KUKA KRL program: MyProgram_268().src

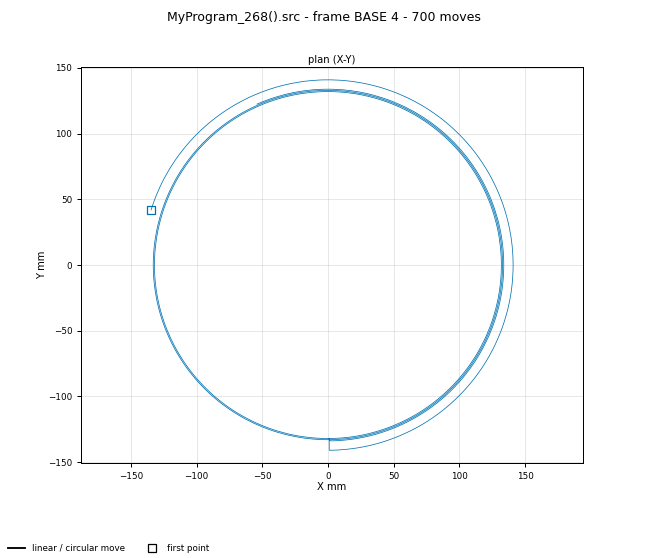
[picture p0: tool path of MyProgram_268().src in frame BASE 4, 700 of 700 moves have a stored position in this frame; points joined in program order, loops and branches not executed]
&ACCESS RVP
&REL 1
&PARAM TEMPLATE = C:\KRC\Roboter\Template\vorgabe
&PARAM EDITMASK = *
DEF MyProgram_268()
; ---- Setting reference (Base) ----
$BASE = BASE_DATA[4]

; --------------------------
; ---- Setting tool (TCP) ----
$TOOL = TOOL_DATA[3]
; --------------------------

$VEL.CP = VEL_APROX_PRINT
Startdeposition()
$VEL.CP = VEL_PRINT
LIN {X -134.5942,Y 41.9312,Z 169,A 163.5765,B 9.595,C 0.2023,E1 9.4446,E2 287.9092} C_DIS
LIN {X -133.5256,Y 45.2188,Z 169,A 161.9808,B 9.595,C 0.2018,E1 9.446,E2 289.5276} C_DIS
LIN {X -132.144,Y 49.1059,Z 169,A 160.3051,B 9.5951,C 0.1972,E1 9.4476,E2 291.2013} C_DIS
LIN {X -130.5039,Y 53.3146,Z 169,A 158.5648,B 9.5953,C 0.1905,E1 9.4494,E2 292.9277} C_DIS
LIN {X -129.1483,Y 56.5189,Z 169,A 157.1411,B 9.5953,C 0.1868,E1 9.451,E2 294.3512} C_DIS
LIN {X -127.8004,Y 59.5017,Z 169,A 155.7818,B 9.5953,C 0.1838,E1 9.4525,E2 295.7126} C_DIS
LIN {X -126.3044,Y 62.6142,Z 169,A 154.3586,B 9.5955,C 0.1804,E1 9.4543,E2 297.1368} C_DIS
LIN {X -124.5762,Y 65.9871,Z 169,A 152.7987,B 9.5955,C 0.1768,E1 9.4563,E2 298.6975} C_DIS
LIN {X -122.6643,Y 69.4801,Z 169,A 151.0806,B 9.5955,C 0.1745,E1 9.4586,E2 300.4266} C_DIS
LIN {X -120.481,Y 73.2001,Z 169,A 149.3244,B 9.5956,C 0.1701,E1 9.4612,E2 302.1813} C_DIS
LIN {X -118.1952,Y 76.8358,Z 169,A 147.5146,B 9.5957,C 0.167,E1 9.4639,E2 303.9974} C_DIS
LIN {X -115.5599,Y 80.7454,Z 169,A 145.5711,B 9.5957,C 0.1628,E1 9.467,E2 305.9422} C_DIS
LIN {X -113.0324,Y 84.2467,Z 169,A 143.81,B 9.5958,C 0.1587,E1 9.4699,E2 307.7022} C_DIS
LIN {X -110.5027,Y 87.5391,Z 169,A 142.0533,B 9.5958,C 0.1561,E1 9.4729,E2 309.466} C_DIS
LIN {X -107.5268,Y 91.1694,Z 169,A 140.2431,B 9.596,C 0.15,E1 9.4761,E2 311.2619} C_DIS
LIN {X -104.992,Y 94.0771,Z 169,A 138.5981,B 9.596,C 0.1479,E1 9.4792,E2 312.915} C_DIS
LIN {X -102.0667,Y 97.2434,Z 169,A 136.8251,B 9.596,C 0.1446,E1 9.4825,E2 314.6888} C_DIS
LIN {X -99.0916,Y 100.2738,Z 169,A 135.045,B 9.5961,C 0.142,E1 9.4861,E2 316.474} C_DIS
LIN {X -95.7403,Y 103.4786,Z 169,A 133.1345,B 9.5961,C 0.1386,E1 9.4899,E2 318.3859} C_DIS
LIN {X -92.5309,Y 106.3574,Z 169,A 131.3797,B 9.5961,C 0.1352,E1 9.4936,E2 320.1393} C_DIS
LIN {X -89.2875,Y 109.0944,Z 169,A 129.6507,B 9.5962,C 0.1321,E1 9.4973,E2 321.8672} C_DIS
LIN {X -85.7732,Y 111.8785,Z 169,A 127.7709,B 9.5962,C 0.1298,E1 9.5015,E2 323.7525} C_DIS
LIN {X -81.9982,Y 114.674,Z 169,A 125.8885,B 9.5963,C 0.126,E1 9.5057,E2 325.6297} C_DIS
LIN {X -78.322,Y 117.2156,Z 169,A 124.0447,B 9.5963,C 0.1235,E1 9.51,E2 327.4753} C_DIS
LIN {X -74.6865,Y 119.5651,Z 169,A 122.2899,B 9.5963,C 0.1206,E1 9.5141,E2 329.2279} C_DIS
LIN {X -70.9951,Y 121.7937,Z 169,A 120.4792,B 9.5964,C 0.1191,E1 9.5185,E2 331.0444} C_DIS
LIN {X -67.2172,Y 123.9185,Z 169,A 118.6942,B 9.5964,C 0.117,E1 9.5228,E2 332.8309} C_DIS
LIN {X -63.389,Y 125.9186,Z 169,A 117.039,B 9.5964,C 0.1126,E1 9.5269,E2 334.4719} C_DIS
LIN {X -60.2838,Y 127.434,Z 169,A 115.6266,B 9.5965,C 0.111,E1 9.5305,E2 335.8842} C_DIS
LIN {X -57.1208,Y 128.8826,Z 169,A 114.2055,B 9.5965,C 0.1094,E1 9.5341,E2 337.305} C_DIS
LIN {X -53.3354,Y 130.4955,Z 169,A 112.4278,B 9.5965,C 0.1095,E1 9.5387,E2 339.0947} C_DIS
LIN {X -49.779,Y 131.8919,Z 169,A 110.9649,B 9.5965,C 0.1061,E1 9.5425,E2 340.5449} C_DIS
LIN {X -46.5347,Y 133.0713,Z 169,A 109.5024,B 9.5965,C 0.1058,E1 9.5463,E2 342.0139} C_DIS
LIN {X -42.5768,Y 134.3899,Z 169,A 107.8494,B 9.5965,C 0.1034,E1 9.5507,E2 343.6603} C_DIS
LIN {X -39.2696,Y 135.3933,Z 169,A 106.4388,B 9.5966,C 0.1023,E1 9.5545,E2 345.0706} C_DIS
LIN {X -35.282,Y 136.4877,Z 169,A 104.6517,B 9.5966,C 0.1032,E1 9.5593,E2 346.87} C_DIS
LIN {X -31.7318,Y 137.3556,Z 169,A 103.2097,B 9.5966,C 0.1012,E1 9.5632,E2 348.3056} C_DIS
LIN {X -27.4911,Y 138.2678,Z 169,A 101.5074,B 9.5966,C 0.0989,E1 9.5679,E2 349.9991} C_DIS
LIN {X -24.1085,Y 138.8981,Z 169,A 100.0991,B 9.5966,C 0.0984,E1 9.5717,E2 351.4079} C_DIS
LIN {X -20.708,Y 139.4459,Z 169,A 98.674,B 9.5966,C 0.0982,E1 9.5757,E2 352.8352} C_DIS
LIN {X -17.26,Y 139.9135,Z 169,A 97.1242,B 9.5966,C 0.1004,E1 9.58,E2 354.4012} C_DIS
LIN {X -12.7769,Y 140.3946,Z 169,A 95.4449,B 9.5966,C 0.0967,E1 9.5846,E2 356.0603} C_DIS
LIN {X -9.3326,Y 140.6654,Z 169,A 94.0962,B 9.5966,C 0.0952,E1 9.5884,E2 357.4014} C_DIS
LIN {X -6.258,Y 140.8362,Z 169,A 92.7456,B 9.5966,C 0.097,E1 9.5922,E2 358.7638} C_DIS
LIN {X -2.4077,Y 140.9526,Z 169,A 91.1279,B 9.5966,C 0.0979,E1 9.5967,E2 360.3872} C_DIS
LIN {X 2.3955,Y 140.9528,Z 169,A 89.2128,B 9.5966,C 0.0972,E1 9.602,E2 362.2968} C_DIS
LIN {X 6.234,Y 140.8372,Z 169,A 87.6868,B 9.5966,C 0.0965,E1 9.6063,E2 363.8178} C_DIS
LIN {X 9.3191,Y 140.6662,Z 169,A 86.4564,B 9.5966,C 0.0962,E1 9.6097,E2 365.0445} C_DIS
LIN {X 12.7648,Y 140.3957,Z 169,A 84.9273,B 9.5966,C 0.0991,E1 9.614,E2 366.5887} C_DIS
LIN {X 17.2433,Y 139.9155,Z 169,A 83.2176,B 9.5966,C 0.0971,E1 9.6187,E2 368.2825} C_DIS
LIN {X 20.6777,Y 139.4502,Z 169,A 81.8119,B 9.5966,C 0.0976,E1 9.6226,E2 369.6875} C_DIS
LIN {X 23.453,Y 139.0086,Z 169,A 80.6674,B 9.5966,C 0.0981,E1 9.6257,E2 370.8318} C_DIS
LIN {X 26.8316,Y 138.3964,Z 169,A 79.1656,B 9.5966,C 0.1011,E1 9.6299,E2 372.3466} C_DIS
LIN {X 31.5211,Y 137.4037,Z 169,A 77.3288,B 9.5966,C 0.0999,E1 9.6349,E2 374.169} C_DIS
LIN {X 35.2505,Y 136.4957,Z 169,A 75.782,B 9.5966,C 0.1006,E1 9.6391,E2 375.7137} C_DIS
LIN {X 38.615,Y 135.5827,Z 169,A 74.3639,B 9.5966,C 0.1017,E1 9.6429,E2 377.1318} C_DIS
LIN {X 41.9329,Y 134.5936,Z 169,A 72.9765,B 9.5966,C 0.1024,E1 9.6466,E2 378.5164} C_DIS
LIN {X 45.2213,Y 133.5247,Z 169,A 71.4108,B 9.5966,C 0.1072,E1 9.6508,E2 380.1023} C_DIS
LIN {X 49.1122,Y 132.1417,Z 169,A 69.7678,B 9.5966,C 0.1081,E1 9.6551,E2 381.7406} C_DIS
LIN {X 53.3187,Y 130.5023,Z 169,A 68.0634,B 9.5966,C 0.1071,E1 9.6594,E2 383.4284} C_DIS
LIN {X 56.5128,Y 129.1509,Z 169,A 66.6736,B 9.5966,C 0.1082,E1 9.663,E2 384.8156} C_DIS
LIN {X 59.4777,Y 127.8115,Z 169,A 65.3498,B 9.5966,C 0.1098,E1 9.6664,E2 386.1396} C_DIS
LIN {X 62.5803,Y 126.3212,Z 169,A 63.9205,B 9.5965,C 0.1122,E1 9.67,E2 387.5727} C_DIS
LIN {X 66.4245,Y 124.3453,Z 169,A 62.2133,B 9.5965,C 0.1134,E1 9.6742,E2 389.2738} C_DIS
LIN {X 69.7802,Y 122.4931,Z 169,A 60.5878,B 9.5965,C 0.1171,E1 9.6782,E2 390.9079} C_DIS
LIN {X 73.5011,Y 120.2975,Z 169,A 58.8315,B 9.5965,C 0.1197,E1 9.6824,E2 392.6644} C_DIS
LIN {X 77.5895,Y 117.7018,Z 169,A 56.8943,B 9.5964,C 0.1221,E1 9.6869,E2 394.598} C_DIS
LIN {X 81.1458,Y 115.2788,Z 169,A 55.1544,B 9.5964,C 0.1247,E1 9.6909,E2 396.3371} C_DIS
LIN {X 84.6708,Y 112.7155,Z 169,A 53.4186,B 9.5964,C 0.1269,E1 9.6948,E2 398.0687} C_DIS
LIN {X 88.0894,Y 110.0647,Z 169,A 51.6799,B 9.5963,C 0.1296,E1 9.6986,E2 399.8054} C_DIS
LIN {X 91.4161,Y 107.317,Z 169,A 49.9188,B 9.5963,C 0.1329,E1 9.7024,E2 401.5679} C_DIS
LIN {X 94.6711,Y 104.4568,Z 169,A 48.1785,B 9.5962,C 0.1358,E1 9.706,E2 403.306} C_DIS
LIN {X 97.836,Y 101.4989,Z 169,A 46.4418,B 9.5962,C 0.1387,E1 9.7095,E2 405.0403} C_DIS
LIN {X 100.8967,Y 98.4571,Z 169,A 44.7252,B 9.5962,C 0.1414,E1 9.7129,E2 406.7527} C_DIS
LIN {X 103.8624,Y 95.3229,Z 169,A 43.0024,B 9.5961,C 0.1444,E1 9.7161,E2 408.4723} C_DIS
LIN {X 106.7472,Y 92.0808,Z 169,A 41.2219,B 9.5961,C 0.1486,E1 9.7194,E2 410.2556} C_DIS
LIN {X 109.5218,Y 88.7632,Z 169,A 39.4703,B 9.5959,C 0.1524,E1 9.7225,E2 412.0072} C_DIS
LIN {X 112.187,Y 85.3699,Z 169,A 37.7746,B 9.5959,C 0.155,E1 9.7254,E2 413.6964} C_DIS
LIN {X 114.7571,Y 81.882,Z 169,A 36.0512,B 9.5959,C 0.1582,E1 9.7282,E2 415.4159} C_DIS
LIN {X 117.2128,Y 78.3262,Z 169,A 34.2819,B 9.5958,C 0.1627,E1 9.731,E2 417.1878} C_DIS
LIN {X 119.555,Y 74.7028,Z 169,A 32.5697,B 9.5958,C 0.1659,E1 9.7336,E2 418.8957} C_DIS
LIN {X 121.7798,Y 71.0191,Z 169,A 30.7924,B 9.5956,C 0.171,E1 9.7361,E2 420.6776} C_DIS
LIN {X 123.9192,Y 67.2159,Z 169,A 29.0406,B 9.5956,C 0.1749,E1 9.7385,E2 422.4277} C_DIS
LIN {X 125.7674,Y 63.686,Z 169,A 27.522,B 9.5956,C 0.1766,E1 9.7404,E2 423.9344} C_DIS
LIN {X 127.4446,Y 60.2617,Z 169,A 26.0271,B 9.5955,C 0.1793,E1 9.7422,E2 425.4234} C_DIS
LIN {X 128.8415,Y 57.2127,Z 169,A 24.6768,B 9.5955,C 0.1826,E1 9.7438,E2 426.7729} C_DIS
LIN {X 130.4933,Y 53.341,Z 169,A 22.9043,B 9.5953,C 0.1887,E1 9.7457,E2 428.5546} C_DIS
LIN {X 131.8908,Y 49.782,Z 169,A 21.4593,B 9.5953,C 0.1902,E1 9.7471,E2 429.9867} C_DIS
LIN {X 133.3051,Y 45.8604,Z 169,A 19.7974,B 9.5952,C 0.194,E1 9.7487,E2 431.6457} C_DIS
LIN {X 134.3891,Y 42.5794,Z 169,A 18.4143,B 9.5952,C 0.1974,E1 9.7499,E2 433.0272} C_DIS
LIN {X 135.3924,Y 39.2725,Z 169,A 17.0291,B 9.5951,C 0.2008,E1 9.751,E2 434.411} C_DIS
LIN {X 136.4894,Y 35.2754,Z 169,A 15.2736,B 9.5949,C 0.2073,E1 9.7522,E2 436.177} C_DIS
LIN {X 137.4032,Y 31.5233,Z 169,A 13.8229,B 9.5949,C 0.2088,E1 9.7532,E2 437.6137} C_DIS
LIN {X 138.267,Y 27.495,Z 169,A 12.1816,B 9.5949,C 0.2127,E1 9.7541,E2 439.2522} C_DIS
LIN {X 138.8977,Y 24.1109,Z 169,A 10.8273,B 9.5947,C 0.2156,E1 9.7548,E2 440.6019} C_DIS
LIN {X 139.3437,Y 21.3717,Z 169,A 9.6887,B 9.5947,C 0.2191,E1 9.7553,E2 441.7429} C_DIS
LIN {X 139.8288,Y 17.9286,Z 169,A 8.1786,B 9.5945,C 0.2256,E1 9.7558,E2 443.2667} C_DIS
LIN {X 140.295,Y 13.8137,Z 169,A 6.6283,B 9.5945,C 0.2272,E1 9.7563,E2 444.8015} C_DIS
LIN {X 140.5909,Y 10.374,Z 169,A 5.2517,B 9.5944,C 0.2306,E1 9.7566,E2 446.1759} C_DIS
LIN {X 140.8029,Y 6.9279,Z 169,A 3.8772,B 9.5944,C 0.234,E1 9.7568,E2 447.548} C_DIS
LIN {X 140.931,Y 3.4756,Z 169,A 2.5047,B 9.5942,C 0.2373,E1 9.7569,E2 448.9178} C_DIS
LIN {X 140.9775,Y -0.0022,Z 169,A 0.8866,B 9.594,C 0.2465,E1 9.7569,E2 450.5638} C_DIS
LIN {X 140.9022,Y -4.5117,Z 169,A -0.6897,B 9.594,C 0.2455,E1 9.7569,E2 452.1086} C_DIS
LIN {X 140.7496,Y -7.9654,Z 169,A -2.0369,B 9.594,C 0.2481,E1 9.7567,E2 453.4496} C_DIS
LIN {X 140.5425,Y -11.0367,Z 169,A -3.3352,B 9.5938,C 0.2529,E1 9.7564,E2 454.7554} C_DIS
LIN {X 140.1868,Y -14.8698,Z 169,A -4.87,B 9.5938,C 0.2567,E1 9.756,E2 456.2878} C_DIS
LIN {X 139.693,Y -18.9651,Z 169,A -6.5053,B 9.5936,C 0.2606,E1 9.7554,E2 457.9195} C_DIS
LIN {X 139.1873,Y -22.3816,Z 169,A -7.9131,B 9.5936,C 0.2648,E1 9.7548,E2 459.3294} C_DIS
LIN {X 138.5947,Y -25.7943,Z 169,A -9.2934,B 9.5934,C 0.2681,E1 9.7541,E2 460.7075} C_DIS
LIN {X 137.8647,Y -29.4408,Z 169,A -10.8555,B 9.5933,C 0.2737,E1 9.7532,E2 462.2777} C_DIS
LIN {X 137.0081,Y -33.1984,Z 169,A -12.3595,B 9.5932,C 0.2767,E1 9.7523,E2 463.7752} C_DIS
LIN {X 136.0578,Y -36.9049,Z 169,A -13.8478,B 9.5932,C 0.2794,E1 9.7512,E2 465.2565} C_DIS
LIN {X 135.1126,Y -40.2284,Z 169,A -15.2331,B 9.593,C 0.2829,E1 9.7501,E2 466.6408} C_DIS
LIN {X 134.1854,Y -43.2169,Z 169,A -16.5209,B 9.5929,C 0.2869,E1 9.749,E2 467.9321} C_DIS
LIN {X 132.7343,Y -47.487,Z 169,A -18.2601,B 9.5929,C 0.2897,E1 9.7475,E2 469.661} C_DIS
LIN {X 131.2801,Y -51.3705,Z 169,A -19.9923,B 9.5926,C 0.2955,E1 9.7457,E2 471.4011} C_DIS
LIN {X 129.8366,Y -54.9196,Z 169,A -21.4938,B 9.5926,C 0.2984,E1 9.7441,E2 472.8971} C_DIS
LIN {X 128.532,Y -57.9047,Z 169,A -22.7978,B 9.5925,C 0.3015,E1 9.7427,E2 474.1998} C_DIS
LIN {X 127.0634,Y -61.0594,Z 169,A -24.1927,B 9.5923,C 0.3048,E1 9.741,E2 475.5938} C_DIS
LIN {X 125.3754,Y -64.4561,Z 169,A -25.7756,B 9.5922,C 0.3099,E1 9.739,E2 477.1837} C_DIS
LIN {X 123.2498,Y -68.435,Z 169,A -27.5651,B 9.5921,C 0.3136,E1 9.7366,E2 478.9695} C_DIS
LIN {X 121.0914,Y -72.1853,Z 169,A -29.3064,B 9.5919,C 0.3177,E1 9.7342,E2 480.7104} C_DIS
LIN {X 118.9256,Y -75.7012,Z 169,A -31.0146,B 9.5918,C 0.3227,E1 9.7316,E2 482.4243} C_DIS
LIN {X 116.4553,Y -79.4491,Z 169,A -32.8335,B 9.5916,C 0.327,E1 9.7288,E2 484.2444} C_DIS
LIN {X 113.7961,Y -83.2128,Z 169,A -34.6594,B 9.5916,C 0.3305,E1 9.7258,E2 486.0662} C_DIS
LIN {X 111.1913,Y -86.663,Z 169,A -36.4151,B 9.5914,C 0.3346,E1 9.7228,E2 487.8235} C_DIS
LIN {X 108.4264,Y -90.0977,Z 169,A -38.158,B 9.5913,C 0.3376,E1 9.7198,E2 489.5619} C_DIS
LIN {X 105.6201,Y -93.3715,Z 169,A -39.8759,B 9.5911,C 0.3407,E1 9.7166,E2 491.277} C_DIS
LIN {X 102.7099,Y -96.5637,Z 169,A -41.6013,B 9.5911,C 0.3439,E1 9.7133,E2 493.0003} C_DIS
LIN {X 99.6849,Y -99.6843,Z 169,A -43.3281,B 9.5909,C 0.3467,E1 9.71,E2 494.7238} C_DIS
LIN {X 96.5855,Y -102.6894,Z 169,A -45.0601,B 9.5909,C 0.3499,E1 9.7065,E2 496.4546} C_DIS
LIN {X 93.3954,Y -105.5989,Z 169,A -46.8058,B 9.5907,C 0.3532,E1 9.7029,E2 498.2008} C_DIS
LIN {X 90.0987,Y -108.4256,Z 169,A -48.5608,B 9.5906,C 0.3565,E1 9.6991,E2 499.9563} C_DIS
LIN {X 86.7378,Y -111.1331,Z 169,A -50.3042,B 9.5905,C 0.3595,E1 9.6953,E2 501.7} C_DIS
LIN {X 83.2951,Y -113.7356,Z 169,A -52.0622,B 9.5903,C 0.3629,E1 9.6914,E2 503.4602} C_DIS
LIN {X 79.773,Y -116.2329,Z 169,A -53.7663,B 9.5903,C 0.3647,E1 9.6875,E2 505.1593} C_DIS
LIN {X 76.1662,Y -118.6279,Z 169,A -55.5425,B 9.5901,C 0.3681,E1 9.6833,E2 506.9393} C_DIS
LIN {X 72.5117,Y -120.8968,Z 169,A -57.2905,B 9.5901,C 0.3709,E1 9.6791,E2 508.6889} C_DIS
LIN {X 68.7803,Y -123.0578,Z 169,A -58.998,B 9.59,C 0.3726,E1 9.675,E2 510.392} C_DIS
LIN {X 65.3914,Y -124.889,Z 169,A -60.5053,B 9.59,C 0.3735,E1 9.6713,E2 511.893} C_DIS
LIN {X 61.8369,Y -126.6879,Z 169,A -62.0901,B 9.5899,C 0.375,E1 9.6673,E2 513.4747} C_DIS
LIN {X 58.733,Y -128.1559,Z 169,A -63.4717,B 9.5899,C 0.3766,E1 9.6639,E2 514.8557} C_DIS
LIN {X 55.6106,Y -129.541,Z 169,A -64.8591,B 9.5898,C 0.3783,E1 9.6603,E2 516.2441} C_DIS
LIN {X 51.8495,Y -131.0939,Z 169,A -66.6301,B 9.5896,C 0.383,E1 9.6557,E2 518.0318} C_DIS
LIN {X 47.5078,Y -132.7268,Z 169,A -68.3666,B 9.5896,C 0.3817,E1 9.6512,E2 519.7503} C_DIS
LIN {X 44.2426,Y -133.8506,Z 169,A -69.762,B 9.5896,C 0.383,E1 9.6475,E2 521.1456} C_DIS
LIN {X 40.9236,Y -134.9026,Z 169,A -71.1692,B 9.5896,C 0.3842,E1 9.6437,E2 522.5528} C_DIS
LIN {X 37.6033,Y -135.8656,Z 169,A -72.6736,B 9.5894,C 0.3877,E1 9.6396,E2 524.0714} C_DIS
LIN {X 33.2171,Y -137.0036,Z 169,A -74.4025,B 9.5894,C 0.3867,E1 9.635,E2 525.7867} C_DIS
LIN {X 29.857,Y -137.7749,Z 169,A -75.8844,B 9.5894,C 0.3896,E1 9.6309,E2 527.2801} C_DIS
LIN {X 25.821,Y -138.5896,Z 169,A -77.4557,B 9.5894,C 0.3884,E1 9.6266,E2 528.8392} C_DIS
LIN {X 22.4208,Y -139.1808,Z 169,A -78.8725,B 9.5894,C 0.3896,E1 9.6227,E2 530.2587} C_DIS
LIN {X 18.9812,Y -139.6909,Z 169,A -80.2838,B 9.5893,C 0.3903,E1 9.6188,E2 531.6707} C_DIS
LIN {X 14.868,Y -140.187,Z 169,A -81.982,B 9.5893,C 0.3914,E1 9.6141,E2 533.3717} C_DIS
LIN {X 11.1093,Y -140.5367,Z 169,A -83.5081,B 9.5893,C 0.3918,E1 9.6099,E2 534.8976} C_DIS
LIN {X 7.9782,Y -140.7489,Z 169,A -84.7464,B 9.5893,C 0.3914,E1 9.6064,E2 536.1317} C_DIS
LIN {X 4.5253,Y -140.9018,Z 169,A -86.2616,B 9.5891,C 0.3941,E1 9.6022,E2 537.6621} C_DIS
LIN {X 1.0246,Y -140.9657,Z 169,A -87.164,B 9.5896,C 0.3829,E1 9.5998,E2 538.4966} C_DIS
Enddeposition()
LIN {X 0.9572,Y -132.0209,Z 170,A -87.7415,B 9.9605,C 0.3252,E1 9.9679,E2 538.6917} C_DIS
Startdeposition()
$VEL.CP = VEL_PRINT
LIN {X 3.7904,Y -131.9708,Z 170,A -86.115,B 9.9607,C 0.3165,E1 9.9726,E2 537.0162} C_DIS
LIN {X 8.0863,Y -131.7772,Z 170,A -84.3027,B 9.9607,C 0.3172,E1 9.9776,E2 535.2096} C_DIS
LIN {X 11.8723,Y -131.4923,Z 170,A -82.5093,B 9.9608,C 0.3134,E1 9.9827,E2 533.3975} C_DIS
LIN {X 16.16,Y -131.0333,Z 170,A -80.6725,B 9.9608,C 0.3134,E1 9.9878,E2 531.5638} C_DIS
LIN {X 19.3657,Y -130.5988,Z 170,A -79.4051,B 9.9608,C 0.3155,E1 9.9912,E2 530.3123} C_DIS
LIN {X 23.1047,Y -129.9876,Z 170,A -77.7513,B 9.9608,C 0.3143,E1 9.9958,E2 528.6562} C_DIS
LIN {X 26.3031,Y -129.3782,Z 170,A -76.2726,B 9.9608,C 0.3119,E1 9.9999,E2 527.1686} C_DIS
LIN {X 30.5034,Y -128.4535,Z 170,A -74.482,B 9.9608,C 0.3121,E1 10.0047,E2 525.386} C_DIS
LIN {X 33.6448,Y -127.6665,Z 170,A -73.0844,B 9.9609,C 0.3111,E1 10.0085,E2 523.9884} C_DIS
LIN {X 36.7643,Y -126.8032,Z 170,A -71.5383,B 9.9611,C 0.3067,E1 10.0127,E2 522.4238} C_DIS
LIN {X 41.3922,Y -125.3688,Z 170,A -69.4899,B 9.9611,C 0.3058,E1 10.0181,E2 520.3805} C_DIS
LIN {X 44.9083,Y -124.1523,Z 170,A -67.937,B 9.9611,C 0.3054,E1 10.0222,E2 518.834} C_DIS
LIN {X 48.7091,Y -122.7128,Z 170,A -66.077,B 9.9612,C 0.3012,E1 10.0271,E2 516.9609} C_DIS
LIN {X 52.0153,Y -121.3469,Z 170,A -64.698,B 9.9612,C 0.3031,E1 10.0306,E2 515.6017} C_DIS
LIN {X 54.9745,Y -120.0355,Z 170,A -63.3038,B 9.9612,C 0.3015,E1 10.0341,E2 514.2077} C_DIS
LIN {X 57.9001,Y -118.6524,Z 170,A -61.8704,B 9.9612,C 0.2989,E1 10.0377,E2 512.7696} C_DIS
LIN {X 60.8063,Y -117.19,Z 170,A -60.4164,B 9.9614,C 0.2959,E1 10.0414,E2 511.3092} C_DIS
LIN {X 64.1291,Y -115.4059,Z 170,A -58.8145,B 9.9614,C 0.2943,E1 10.0453,E2 509.7102} C_DIS
LIN {X 67.8372,Y -113.2661,Z 170,A -57.0334,B 9.9614,C 0.2931,E1 10.0496,E2 507.9367} C_DIS
LIN {X 70.629,Y -111.5464,Z 170,A -55.5169,B 9.9616,C 0.2886,E1 10.0532,E2 506.4074} C_DIS
LIN {X 73.8128,Y -109.4657,Z 170,A -53.8877,B 9.9616,C 0.2862,E1 10.057,E2 504.7793} C_DIS
LIN {X 77.3447,Y -106.9993,Z 170,A -52.1417,B 9.9616,C 0.2857,E1 10.0609,E2 503.0466} C_DIS
LIN {X 80.1576,Y -104.9084,Z 170,A -50.5419,B 9.9618,C 0.2811,E1 10.0645,E2 501.4358} C_DIS
LIN {X 83.542,Y -102.2338,Z 170,A -48.6838,B 9.9618,C 0.2778,E1 10.0685,E2 499.5775} C_DIS
LIN {X 86.8446,Y -99.4436,Z 170,A -46.8696,B 9.962,C 0.2755,E1 10.0724,E2 497.7691} C_DIS
LIN {X 89.847,Y -96.7397,Z 170,A -45.1313,B 9.962,C 0.2723,E1 10.076,E2 496.0308} C_DIS
LIN {X 92.7363,Y -93.9743,Z 170,A -43.3386,B 9.9622,C 0.2673,E1 10.0796,E2 494.2294} C_DIS
LIN {X 95.6179,Y -91.0401,Z 170,A -41.661,B 9.9622,C 0.2659,E1 10.0828,E2 492.5631} C_DIS
LIN {X 98.3647,Y -88.0648,Z 170,A -39.8809,B 9.9623,C 0.2614,E1 10.0861,E2 490.7784} C_DIS
LIN {X 100.996,Y -85.0345,Z 170,A -38.1028,B 9.9625,C 0.2566,E1 10.0894,E2 488.9939} C_DIS
LIN {X 103.9098,Y -81.4481,Z 170,A -36.2159,B 9.9625,C 0.2547,E1 10.0926,E2 487.1194} C_DIS
LIN {X 106.375,Y -78.2009,Z 170,A -34.5164,B 9.9625,C 0.2521,E1 10.0955,E2 485.4266} C_DIS
LIN {X 108.2546,Y -75.5778,Z 170,A -33.0352,B 9.9627,C 0.2467,E1 10.0979,E2 483.934} C_DIS
LIN {X 110.6681,Y -71.9972,Z 170,A -31.1834,B 9.9628,C 0.2426,E1 10.1007,E2 482.0829} C_DIS
LIN {X 112.694,Y -68.7836,Z 170,A -29.5428,B 9.9628,C 0.2386,E1 10.1031,E2 480.4414} C_DIS
LIN {X 114.8835,Y -65.0613,Z 170,A -27.7988,B 9.9629,C 0.2368,E1 10.1056,E2 478.7113} C_DIS
LIN {X 116.4391,Y -62.2338,Z 170,A -26.2814,B 9.9631,C 0.2304,E1 10.1076,E2 477.1781} C_DIS
LIN {X 118.172,Y -58.8739,Z 170,A -24.8109,B 9.9631,C 0.2301,E1 10.1094,E2 475.7266} C_DIS
LIN {X 119.5747,Y -55.9711,Z 170,A -23.4316,B 9.9631,C 0.2268,E1 10.1111,E2 474.3482} C_DIS
LIN {X 120.9038,Y -53.0403,Z 170,A -22.0317,B 9.9633,C 0.2229,E1 10.1127,E2 472.9464} C_DIS
LIN {X 122.3784,Y -49.5386,Z 170,A -20.6011,B 9.9633,C 0.2236,E1 10.1142,E2 471.5404} C_DIS
LIN {X 123.3769,Y -47.0023,Z 170,A -19.1123,B 9.9635,C 0.2131,E1 10.1157,E2 470.0132} C_DIS
LIN {X 124.8489,Y -42.9345,Z 170,A -17.403,B 9.9635,C 0.2119,E1 10.1173,E2 468.3223} C_DIS
LIN {X 126.0377,Y -39.3132,Z 170,A -15.6421,B 9.9636,C 0.2046,E1 10.1188,E2 466.5467} C_DIS
LIN {X 126.9502,Y -36.2591,Z 170,A -14.2692,B 9.9637,C 0.201,E1 10.1199,E2 465.1736} C_DIS
LIN {X 127.7953,Y -33.1572,Z 170,A -13.0332,B 9.9637,C 0.2008,E1 10.1207,E2 463.9554} C_DIS
LIN {X 128.5625,Y -30.0449,Z 170,A -11.6609,B 9.9637,C 0.1973,E1 10.1216,E2 462.584} C_DIS
LIN {X 129.1832,Y -27.2518,Z 170,A -10.4504,B 9.9638,C 0.1945,E1 10.1223,E2 461.3759} C_DIS
LIN {X 129.798,Y -24.1552,Z 170,A -8.9542,B 9.964,C 0.1875,E1 10.1231,E2 459.8629} C_DIS
LIN {X 130.4371,Y -20.4158,Z 170,A -7.6519,B 9.964,C 0.191,E1 10.1237,E2 458.6006} C_DIS
LIN {X 130.8978,Y -17.2154,Z 170,A -6.0843,B 9.964,C 0.183,E1 10.1243,E2 457.0117} C_DIS
LIN {X 131.3219,Y -13.6174,Z 170,A -4.5427,B 9.9641,C 0.1791,E1 10.1248,E2 455.4723} C_DIS
LIN {X 131.6675,Y -9.7115,Z 170,A -2.7777,B 9.9642,C 0.1726,E1 10.1252,E2 453.6978} C_DIS
LIN {X 131.8945,Y -5.9158,Z 170,A -1.0926,B 9.9643,C 0.167,E1 10.1254,E2 452.0069} C_DIS
LIN {X 132.0165,Y -1.6207,Z 170,A 0.6383,B 9.9643,C 0.1648,E1 10.1255,E2 450.2903} C_DIS
LIN {X 132.0165,Y 1.6169,Z 170,A 2.1229,B 9.9645,C 0.1587,E1 10.1255,E2 448.7948} C_DIS
LIN {X 131.8949,Y 5.9072,Z 170,A 3.9795,B 9.9645,C 0.1535,E1 10.1253,E2 446.9371} C_DIS
LIN {X 131.6354,Y 10.1505,Z 170,A 5.6368,B 9.9645,C 0.1526,E1 10.125,E2 445.3008} C_DIS
LIN {X 131.2812,Y 13.9955,Z 170,A 7.3777,B 9.9647,C 0.1462,E1 10.1245,E2 443.5504} C_DIS
LIN {X 130.7475,Y 18.3254,Z 170,A 8.9852,B 9.9647,C 0.1475,E1 10.1239,E2 441.9757} C_DIS
LIN {X 130.35,Y 20.9772,Z 170,A 10.4606,B 9.9647,C 0.1367,E1 10.1233,E2 440.4617} C_DIS
LIN {X 129.6917,Y 24.7114,Z 170,A 11.9285,B 9.9648,C 0.1363,E1 10.1225,E2 439.0138} C_DIS
LIN {X 128.9396,Y 28.38,Z 170,A 13.6448,B 9.9648,C 0.1295,E1 10.1215,E2 437.285} C_DIS
LIN {X 128.0676,Y 32.0844,Z 170,A 15.1589,B 9.9649,C 0.1281,E1 10.1206,E2 435.7861} C_DIS
LIN {X 127.0143,Y 36.03,Z 170,A 16.8788,B 9.9649,C 0.1244,E1 10.1193,E2 434.0711} C_DIS
LIN {X 126.1728,Y 38.8718,Z 170,A 18.1711,B 9.965,C 0.1207,E1 10.1182,E2 432.777} C_DIS
LIN {X 125.185,Y 41.944,Z 170,A 19.5524,B 9.965,C 0.1173,E1 10.117,E2 431.3969} C_DIS
LIN {X 124.1222,Y 44.9916,Z 170,A 20.988,B 9.965,C 0.1126,E1 10.1157,E2 429.9561} C_DIS
LIN {X 122.5862,Y 49.023,Z 170,A 22.7786,B 9.9651,C 0.1095,E1 10.1139,E2 428.1739} C_DIS
LIN {X 121.3454,Y 52.0189,Z 170,A 24.1665,B 9.9651,C 0.1062,E1 10.1124,E2 426.7873} C_DIS
LIN {X 120.0335,Y 54.979,Z 170,A 25.5508,B 9.9651,C 0.103,E1 10.1108,E2 425.4045} C_DIS
LIN {X 118.6488,Y 57.9073,Z 170,A 26.9357,B 9.9652,C 0.0998,E1 10.1091,E2 424.0212} C_DIS
LIN {X 116.9582,Y 61.2477,Z 170,A 28.4695,B 9.9652,C 0.0978,E1 10.1072,E2 422.4972} C_DIS
LIN {X 115.5299,Y 63.9051,Z 170,A 29.8657,B 9.9652,C 0.0924,E1 10.1053,E2 421.0898} C_DIS
LIN {X 113.7869,Y 66.9596,Z 170,A 31.4345,B 9.9653,C 0.0876,E1 10.1031,E2 419.515} C_DIS
LIN {X 111.5414,Y 70.6369,Z 170,A 33.2989,B 9.9653,C 0.0832,E1 10.1003,E2 417.6501} C_DIS
LIN {X 109.4667,Y 73.8114,Z 170,A 34.9156,B 9.9654,C 0.0799,E1 10.0978,E2 416.036} C_DIS
LIN {X 106.9971,Y 77.3478,Z 170,A 36.669,B 9.9654,C 0.0783,E1 10.095,E2 414.2958} C_DIS
LIN {X 104.5859,Y 80.5789,Z 170,A 38.4585,B 9.9654,C 0.0733,E1 10.092,E2 412.5006} C_DIS
LIN {X 102.0777,Y 83.733,Z 170,A 40.1631,B 9.9654,C 0.0704,E1 10.089,E2 410.8005} C_DIS
LIN {X 99.4407,Y 86.848,Z 170,A 41.9239,B 9.9655,C 0.0668,E1 10.0858,E2 409.0402} C_DIS
LIN {X 96.7272,Y 89.8604,Z 170,A 43.6693,B 9.9655,C 0.0634,E1 10.0825,E2 407.2958} C_DIS
LIN {X 93.9558,Y 92.7551,Z 170,A 45.3154,B 9.9655,C 0.0619,E1 10.0793,E2 405.6601} C_DIS
LIN {X 91.6246,Y 95.058,Z 170,A 46.7926,B 9.9655,C 0.0578,E1 10.0764,E2 404.1758} C_DIS
LIN {X 88.671,Y 97.8186,Z 170,A 48.5674,B 9.9655,C 0.054,E1 10.0727,E2 402.398} C_DIS
LIN {X 85.6209,Y 100.4993,Z 170,A 50.2829,B 9.9655,C 0.0517,E1 10.0691,E2 400.6876} C_DIS
LIN {X 82.5016,Y 103.0758,Z 170,A 52.0308,B 9.9656,C 0.0487,E1 10.0653,E2 398.9402} C_DIS
LIN {X 79.4915,Y 105.4141,Z 170,A 53.6799,B 9.9656,C 0.046,E1 10.0617,E2 397.2913} C_DIS
LIN {X 76.0316,Y 107.9362,Z 170,A 55.4485,B 9.9656,C 0.0449,E1 10.0577,E2 395.5329} C_DIS
LIN {X 73.3744,Y 109.7598,Z 170,A 56.9257,B 9.9656,C 0.0409,E1 10.0542,E2 394.0462} C_DIS
LIN {X 70.1652,Y 111.8391,Z 170,A 58.4879,B 9.9656,C 0.0405,E1 10.0506,E2 392.4954} C_DIS
LIN {X 66.9572,Y 113.7883,Z 170,A 60.193,B 9.9656,C 0.0364,E1 10.0465,E2 390.781} C_DIS
LIN {X 63.6659,Y 115.6624,Z 170,A 61.7352,B 9.9656,C 0.0364,E1 10.0427,E2 389.2508} C_DIS
LIN {X 60.2995,Y 117.4507,Z 170,A 63.3682,B 9.9656,C 0.0347,E1 10.0387,E2 387.6201} C_DIS
LIN {X 57.4018,Y 118.8941,Z 170,A 64.764,B 9.9656,C 0.0331,E1 10.0352,E2 386.2254} C_DIS
LIN {X 54.4729,Y 120.2647,Z 170,A 66.161,B 9.9656,C 0.0316,E1 10.0317,E2 384.8292} C_DIS
LIN {X 51.5089,Y 121.564,Z 170,A 67.6983,B 9.9656,C 0.0272,E1 10.0277,E2 383.2762} C_DIS
LIN {X 48.1124,Y 122.9463,Z 170,A 68.989,B 9.9656,C 0.032,E1 10.0244,E2 382.0212} C_DIS
LIN {X 45.0052,Y 124.1173,Z 170,A 70.6838,B 9.9656,C 0.0251,E1 10.0199,E2 380.2965} C_DIS
LIN {X 41.4138,Y 125.3616,Z 170,A 72.2196,B 9.9656,C 0.0261,E1 10.0159,E2 378.7744} C_DIS
LIN {X 38.3348,Y 126.3372,Z 170,A 73.6795,B 9.9656,C 0.0237,E1 10.012,E2 377.3078} C_DIS
LIN {X 34.2212,Y 127.5128,Z 170,A 75.283,B 9.9656,C 0.0277,E1 10.0077,E2 375.7345} C_DIS
LIN {X 31.601,Y 128.1889,Z 170,A 76.7908,B 9.9657,C 0.0198,E1 10.0035,E2 374.1877} C_DIS
LIN {X 27.34,Y 129.1641,Z 170,A 78.5203,B 9.9657,C 0.0222,E1 9.9989,E2 372.4784} C_DIS
LIN {X 24.1649,Y 129.7962,Z 170,A 80.064,B 9.9657,C 0.0186,E1 9.9946,E2 370.9187} C_DIS
LIN {X 20.4273,Y 130.4353,Z 170,A 81.3808,B 9.9657,C 0.0247,E1 9.9911,E2 369.6411} C_DIS
LIN {X 17.2236,Y 130.8967,Z 170,A 83.0168,B 9.9657,C 0.0194,E1 9.9865,E2 367.9783} C_DIS
LIN {X 14.0026,Y 131.2804,Z 170,A 84.4295,B 9.9657,C 0.0189,E1 9.9826,E2 366.5656} C_DIS
LIN {X 9.712,Y 131.6674,Z 170,A 86.3241,B 9.9657,C 0.018,E1 9.9773,E2 364.6686} C_DIS
LIN {X 5.9272,Y 131.8939,Z 170,A 88.0312,B 9.9657,C 0.0165,E1 9.9725,E2 362.9551} C_DIS
LIN {X 1.6307,Y 132.0163,Z 170,A 89.7313,B 9.9657,C 0.0199,E1 9.9678,E2 361.2753} C_DIS
LIN {X -2.0684,Y 132.009,Z 170,A 91.3831,B 9.9657,C 0.019,E1 9.9632,E2 359.6186} C_DIS
LIN {X -5.9197,Y 131.8943,Z 170,A 93.1883,B 9.9657,C 0.0166,E1 9.9581,E2 357.7987} C_DIS
LIN {X -9.9911,Y 131.647,Z 170,A 94.8151,B 9.9657,C 0.0199,E1 9.9536,E2 356.1896} C_DIS
LIN {X -13.9954,Y 131.2812,Z 170,A 96.6417,B 9.9657,C 0.0188,E1 9.9485,E2 354.3544} C_DIS
LIN {X -18.3198,Y 130.7483,Z 170,A 98.2755,B 9.9657,C 0.0247,E1 9.9441,E2 352.752} C_DIS
LIN {X -20.9696,Y 130.3513,Z 170,A 99.7753,B 9.9657,C 0.0186,E1 9.9398,E2 351.2132} C_DIS
LIN {X -24.7028,Y 129.6933,Z 170,A 101.2999,B 9.9657,C 0.0219,E1 9.9357,E2 349.7038} C_DIS
LIN {X -28.3686,Y 128.9421,Z 170,A 103.0138,B 9.9657,C 0.0212,E1 9.931,E2 347.9804} C_DIS
LIN {X -32.0804,Y 128.0686,Z 170,A 104.5586,B 9.9657,C 0.0245,E1 9.9268,E2 346.4497} C_DIS
LIN {X -35.2287,Y 127.2384,Z 170,A 105.976,B 9.9657,C 0.0256,E1 9.923,E2 345.0327} C_DIS
LIN {X -38.8646,Y 126.175,Z 170,A 107.6261,B 9.9657,C 0.0269,E1 9.9186,E2 343.3831} C_DIS
LIN {X -41.9396,Y 125.1865,Z 170,A 109.035,B 9.9657,C 0.0281,E1 9.9149,E2 341.9743} C_DIS
LIN {X -44.9895,Y 124.123,Z 170,A 110.4999,B 9.9657,C 0.0283,E1 9.911,E2 340.5031} C_DIS
LIN {X -49.0041,Y 122.5939,Z 170,A 112.3169,B 9.9657,C 0.0312,E1 9.9063,E2 338.6931} C_DIS
LIN {X -51.9891,Y 121.3583,Z 170,A 113.7366,B 9.9657,C 0.0325,E1 9.9026,E2 337.2724} C_DIS
LIN {X -54.9774,Y 120.0342,Z 170,A 115.1537,B 9.9657,C 0.0343,E1 9.899,E2 335.8568} C_DIS
LIN {X -58.1652,Y 118.5216,Z 170,A 116.6049,B 9.9657,C 0.0378,E1 9.8954,E2 334.4162} C_DIS
LIN {X -60.8079,Y 117.1892,Z 170,A 118.0828,B 9.9657,C 0.0359,E1 9.8917,E2 332.9167} C_DIS
LIN {X -64.1452,Y 115.397,Z 170,A 119.6513,B 9.9657,C 0.0397,E1 9.8879,E2 331.3585} C_DIS
LIN {X -66.9505,Y 113.7922,Z 170,A 121.153,B 9.9657,C 0.0399,E1 9.8842,E2 329.8464} C_DIS
LIN {X -70.6187,Y 111.5529,Z 170,A 123.0496,B 9.9657,C 0.0423,E1 9.8797,E2 327.9478} C_DIS
LIN {X -74.3844,Y 109.0786,Z 170,A 124.9979,B 9.9657,C 0.0456,E1 9.8752,E2 326.0021} C_DIS
LIN {X -77.568,Y 106.8374,Z 170,A 126.5381,B 9.9656,C 0.0513,E1 9.8717,E2 324.4811} C_DIS
LIN {X -80.4864,Y 104.657,Z 170,A 128.2488,B 9.9656,C 0.0518,E1 9.8679,E2 322.7566} C_DIS
LIN {X -83.7504,Y 102.0635,Z 170,A 130.0911,B 9.9656,C 0.0545,E1 9.8639,E2 320.9122} C_DIS
LIN {X -86.8543,Y 99.4352,Z 170,A 131.8737,B 9.9656,C 0.0576,E1 9.8601,E2 319.1293} C_DIS
LIN {X -89.8575,Y 96.7299,Z 170,A 133.6549,B 9.9656,C 0.0606,E1 9.8564,E2 317.3466} C_DIS
LIN {X -92.7762,Y 93.9348,Z 170,A 135.4913,B 9.9656,C 0.0628,E1 9.8527,E2 315.5023} C_DIS
LIN {X -95.7918,Y 90.8574,Z 170,A 137.3832,B 9.9656,C 0.0664,E1 9.8491,E2 313.6097} C_DIS
LIN {X -98.5534,Y 87.8541,Z 170,A 139.1646,B 9.9655,C 0.0701,E1 9.8457,E2 311.8289} C_DIS
LIN {X -101.3592,Y 84.6017,Z 170,A 141.0576,B 9.9655,C 0.0737,E1 9.8423,E2 309.9344} C_DIS
LIN {X -104.0877,Y 81.2215,Z 170,A 142.9831,B 9.9655,C 0.0774,E1 9.839,E2 308.006} C_DIS
LIN {X -106.4052,Y 78.1598,Z 170,A 144.531,B 9.9654,C 0.0835,E1 9.8364,E2 306.4739} C_DIS
LIN {X -108.2779,Y 75.5444,Z 170,A 146.0424,B 9.9654,C 0.0848,E1 9.834,E2 304.9504} C_DIS
LIN {X -110.6689,Y 71.9961,Z 170,A 147.9259,B 9.9654,C 0.0889,E1 9.8311,E2 303.0657} C_DIS
LIN {X -112.6817,Y 68.8036,Z 170,A 149.591,B 9.9653,C 0.0925,E1 9.8286,E2 301.3991} C_DIS
LIN {X -114.8552,Y 65.111,Z 170,A 151.3764,B 9.9653,C 0.0985,E1 9.8261,E2 299.6245} C_DIS
LIN {X -116.4384,Y 62.2351,Z 170,A 152.9627,B 9.9653,C 0.0994,E1 9.824,E2 298.0207} C_DIS
LIN {X -118.1764,Y 58.8651,Z 170,A 154.4774,B 9.9652,C 0.106,E1 9.8221,E2 296.5231} C_DIS
LIN {X -119.5823,Y 55.9546,Z 170,A 155.9005,B 9.9652,C 0.1094,E1 9.8204,E2 295.0991} C_DIS
LIN {X -120.917,Y 53.0096,Z 170,A 157.3321,B 9.9651,C 0.1127,E1 9.8188,E2 293.6658} C_DIS
LIN {X -122.3782,Y 49.539,Z 170,A 158.9615,B 9.9651,C 0.1172,E1 9.817,E2 292.0386} C_DIS
LIN {X -123.3851,Y 46.9803,Z 170,A 160.3399,B 9.9651,C 0.1172,E1 9.8156,E2 290.6397} C_DIS
LIN {X -124.8459,Y 42.9434,Z 170,A 162.0879,B 9.965,C 0.1244,E1 9.814,E2 288.9073} C_DIS
LIN {X -126.022,Y 39.3646,Z 170,A 163.8995,B 9.965,C 0.1259,E1 9.8125,E2 287.0765} C_DIS
LIN {X -126.9542,Y 36.2449,Z 170,A 165.3248,B 9.9649,C 0.1296,E1 9.8114,E2 285.6513} C_DIS
LIN {X -127.8035,Y 33.125,Z 170,A 166.6093,B 9.9649,C 0.1357,E1 9.8105,E2 284.3823} C_DIS
LIN {X -128.576,Y 29.9856,Z 170,A 168.0915,B 9.9648,C 0.1383,E1 9.8095,E2 282.8922} C_DIS
LIN {X -129.2201,Y 27.0801,Z 170,A 169.3248,B 9.9648,C 0.143,E1 9.8088,E2 281.6672} C_DIS
LIN {X -129.7892,Y 24.2012,Z 170,A 170.7529,B 9.9647,C 0.144,E1 9.808,E2 280.2221} C_DIS
LIN {X -130.4365,Y 20.4196,Z 170,A 172.1308,B 9.9645,C 0.1538,E1 9.8074,E2 278.8799} C_DIS
LIN {X -130.8979,Y 17.2144,Z 170,A 173.7494,B 9.9645,C 0.1542,E1 9.8068,E2 277.2374} C_DIS
LIN {X -131.2807,Y 14.0002,Z 170,A 175.2598,B 9.9645,C 0.1564,E1 9.8063,E2 275.7159} C_DIS
LIN {X -131.6678,Y 9.7074,Z 170,A 177.1552,B 9.9645,C 0.1614,E1 9.8059,E2 273.8196} C_DIS
LIN {X -131.8943,Y 5.9196,Z 170,A 178.8921,B 9.9644,C 0.1647,E1 9.8056,E2 272.0736} C_DIS
LIN {X -132.0165,Y 1.6213,Z 170,A -179.3219,B 9.9643,C 0.1715,E1 9.8056,E2 270.299} C_DIS
LIN {X -132.0164,Y -1.6277,Z 170,A -177.7881,B 9.9643,C 0.1734,E1 9.8056,E2 268.7518} C_DIS
LIN {X -131.8938,Y -5.9283,Z 170,A -175.8763,B 9.9641,C 0.1781,E1 9.8058,E2 266.8365} C_DIS
LIN {X -131.6673,Y -9.7143,Z 170,A -174.2984,B 9.9641,C 0.1841,E1 9.8061,E2 265.2682} C_DIS
LIN {X -131.281,Y -13.997,Z 170,A -172.4401,B 9.9639,C 0.1896,E1 9.8066,E2 263.4125} C_DIS
LIN {X -130.8249,Y -17.772,Z 170,A -170.7983,B 9.9639,C 0.1945,E1 9.8071,E2 261.7733} C_DIS
LIN {X -130.3421,Y -21.0243,Z 170,A -169.189,B 9.9639,C 0.1954,E1 9.8079,E2 260.1435} C_DIS
LIN {X -129.6872,Y -24.7348,Z 170,A -167.6822,B 9.9637,C 0.2023,E1 9.8086,E2 258.6534} C_DIS
LIN {X -128.9384,Y -28.3856,Z 170,A -165.9243,B 9.9637,C 0.2044,E1 9.8096,E2 256.8801} C_DIS
LIN {X -128.0731,Y -32.0628,Z 170,A -164.3753,B 9.9635,C 0.2106,E1 9.8107,E2 255.3433} C_DIS
LIN {X -127.2524,Y -35.1787,Z 170,A -162.9585,B 9.9635,C 0.2142,E1 9.8117,E2 253.9254} C_DIS
LIN {X -126.1765,Y -38.8598,Z 170,A -161.2691,B 9.9634,C 0.2184,E1 9.813,E2 252.2344} C_DIS
LIN {X -125.1866,Y -41.9392,Z 170,A -159.8448,B 9.9633,C 0.2219,E1 9.8143,E2 250.8088} C_DIS
LIN {X -124.0044,Y -45.3183,Z 170,A -158.259,B 9.9632,C 0.2255,E1 9.8158,E2 249.2202} C_DIS
LIN {X -122.5853,Y -49.0255,Z 170,A -156.5236,B 9.9631,C 0.2299,E1 9.8175,E2 247.4846} C_DIS
LIN {X -121.3461,Y -52.0174,Z 170,A -155.1003,B 9.9631,C 0.2333,E1 9.8191,E2 246.0602} C_DIS
LIN {X -120.0277,Y -54.9914,Z 170,A -153.6715,B 9.9629,C 0.2367,E1 9.8207,E2 244.6304} C_DIS
LIN {X -118.6461,Y -57.9129,Z 170,A -152.2518,B 9.9629,C 0.24,E1 9.8224,E2 243.2096} C_DIS
LIN {X -117.1936,Y -60.7994,Z 170,A -150.7328,B 9.9629,C 0.2415,E1 9.8244,E2 241.6774} C_DIS
LIN {X -115.4068,Y -64.1275,Z 170,A -149.1564,B 9.9627,C 0.2467,E1 9.8265,E2 240.1097} C_DIS
LIN {X -113.7887,Y -66.9565,Z 170,A -147.6355,B 9.9627,C 0.2483,E1 9.8286,E2 238.5768} C_DIS
LIN {X -111.5436,Y -70.6334,Z 170,A -145.7929,B 9.9625,C 0.2533,E1 9.8314,E2 236.7386} C_DIS
LIN {X -109.4608,Y -73.8201,Z 170,A -144.0641,B 9.9625,C 0.2558,E1 9.834,E2 235.0015} C_DIS
LIN {X -107.0028,Y -77.3398,Z 170,A -142.2829,B 9.9623,C 0.2617,E1 9.8369,E2 233.2311} C_DIS
LIN {X -104.909,Y -80.1568,Z 170,A -140.6463,B 9.9623,C 0.263,E1 9.8397,E2 231.5816} C_DIS
LIN {X -102.247,Y -83.5258,Z 170,A -138.7521,B 9.9622,C 0.2666,E1 9.843,E2 229.6846} C_DIS
LIN {X -99.4371,Y -86.8521,Z 170,A -136.8937,B 9.9621,C 0.2712,E1 9.8464,E2 227.8307} C_DIS
LIN {X -96.7349,Y -89.8521,Z 170,A -135.1138,B 9.962,C 0.2743,E1 9.8497,E2 226.0482} C_DIS
LIN {X -93.9294,Y -92.7817,Z 170,A -133.2592,B 9.962,C 0.2761,E1 9.8534,E2 224.1829} C_DIS
LIN {X -91.0395,Y -95.6185,Z 170,A -131.5751,B 9.9618,C 0.2809,E1 9.8567,E2 222.5082} C_DIS
LIN {X -88.0743,Y -98.3562,Z 170,A -129.7528,B 9.9618,C 0.2828,E1 9.8605,E2 220.6779} C_DIS
LIN {X -85.0046,Y -101.0211,Z 170,A -127.9573,B 9.9617,C 0.2854,E1 9.8643,E2 218.879} C_DIS
LIN {X -81.8598,Y -103.5864,Z 170,A -126.159,B 9.9617,C 0.2878,E1 9.8683,E2 217.0768} C_DIS
LIN {X -78.2096,Y -106.3686,Z 170,A -124.283,B 9.9615,C 0.2933,E1 9.8724,E2 215.2152} C_DIS
LIN {X -75.5871,Y -108.2482,Z 170,A -122.7697,B 9.9615,C 0.2933,E1 9.8759,E2 213.6884} C_DIS
LIN {X -71.8525,Y -110.7621,Z 170,A -120.8359,B 9.9614,C 0.2967,E1 9.8804,E2 211.7574} C_DIS
LIN {X -68.7857,Y -112.6927,Z 170,A -119.209,B 9.9614,C 0.2979,E1 9.8843,E2 210.124} C_DIS
LIN {X -65.0821,Y -114.8716,Z 170,A -117.2862,B 9.9613,C 0.2993,E1 9.8889,E2 208.1943} C_DIS
LIN {X -61.7702,Y -116.6839,Z 170,A -115.8036,B 9.9611,C 0.3044,E1 9.8925,E2 206.7306} C_DIS
LIN {X -58.9614,Y -118.1288,Z 170,A -114.4444,B 9.9611,C 0.3063,E1 9.8959,E2 205.373} C_DIS
LIN {X -56.238,Y -119.4502,Z 170,A -113.0073,B 9.9611,C 0.3054,E1 9.8996,E2 203.9209} C_DIS
LIN {X -52.9956,Y -120.9231,Z 170,A -111.4019,B 9.9611,C 0.3058,E1 9.9037,E2 202.3081} C_DIS
LIN {X -49.025,Y -122.5854,Z 170,A -109.5779,B 9.961,C 0.3086,E1 9.9084,E2 200.4893} C_DIS
LIN {X -44.9977,Y -124.12,Z 170,A -107.6726,B 9.961,C 0.3095,E1 9.9134,E2 198.5795} C_DIS
LIN {X -41.4231,Y -125.3585,Z 170,A -106.1274,B 9.9609,C 0.3128,E1 9.9175,E2 197.0459} C_DIS
LIN {X -38.3453,Y -126.3339,Z 170,A -104.6625,B 9.9609,C 0.3126,E1 9.9214,E2 195.573} C_DIS
LIN {X -34.2401,Y -127.5077,Z 170,A -102.8587,B 9.9609,C 0.3148,E1 9.9262,E2 193.7749} C_DIS
LIN {X -31.547,Y -128.2019,Z 170,A -101.6395,B 9.9608,C 0.3153,E1 9.9295,E2 192.554} C_DIS
LIN {X -28.3814,Y -128.9393,Z 170,A -100.1116,B 9.9608,C 0.3136,E1 9.9337,E2 191.0113} C_DIS
LIN {X -24.1678,Y -129.7956,Z 170,A -98.2306,B 9.9608,C 0.3141,E1 9.9389,E2 189.128} C_DIS
LIN {X -20.431,Y -130.4347,Z 170,A -96.9033,B 9.9606,C 0.3212,E1 9.9425,E2 187.839} C_DIS
LIN {X -17.2201,Y -130.8972,Z 170,A -95.2606,B 9.9607,C 0.3168,E1 9.9471,E2 186.1672} C_DIS
LIN {X -13.9969,Y -131.281,Z 170,A -93.8472,B 9.9607,C 0.3169,E1 9.951,E2 184.7527} C_DIS
LIN {X -9.7155,Y -131.6672,Z 170,A -91.9519,B 9.9607,C 0.3165,E1 9.9563,E2 182.8529} C_DIS
LIN {X -5.9373,Y -131.8934,Z 170,A -90.2478,B 9.9607,C 0.3153,E1 9.9611,E2 181.1407} C_DIS
LIN {X -1.6378,Y -132.0162,Z 170,A -88.5434,B 9.9607,C 0.3186,E1 9.9658,E2 179.4553} C_DIS
LIN {X 0.9572,Y -132.0209,Z 170,A -87.7409,B 9.9605,C 0.3253,E1 9.9679,E2 178.6917} C_DIS
Enddeposition()
LIN {X 0.9572,Y -132.0209,Z 170,A -87.7409,B 9.9605,C 0.3253,E1 9.9679,E2 178.6917} C_DIS
Startdeposition()
$VEL.CP = VEL_PRINT
LIN {X -0.1872,Y -132.938,Z 170,A -88.8279,B 9.9598,C 0.3438,E1 9.9645,E2 179.8858} C_DIS
LIN {X -3.5112,Y -132.8907,Z 170,A -90.0213,B 9.9599,C 0.3389,E1 9.9612,E2 181.0506} C_DIS
LIN {X -7.9442,Y -132.6995,Z 170,A -91.8892,B 9.9599,C 0.3379,E1 9.956,E2 182.9139} C_DIS
LIN {X -12.0459,Y -132.3916,Z 170,A -93.7466,B 9.9599,C 0.3395,E1 9.9508,E2 184.7824} C_DIS
LIN {X -15.8814,Y -131.9848,Z 170,A -95.2868,B 9.96,C 0.3366,E1 9.9466,E2 186.3083} C_DIS
LIN {X -19.4649,Y -131.5057,Z 170,A -96.8881,B 9.96,C 0.3371,E1 9.9422,E2 187.9154} C_DIS
LIN {X -23.1679,Y -130.9026,Z 170,A -98.5067,B 9.96,C 0.3365,E1 9.9377,E2 189.5346} C_DIS
LIN {X -26.699,Y -130.2281,Z 170,A -99.9912,B 9.96,C 0.3345,E1 9.9336,E2 191.0116} C_DIS
LIN {X -29.5715,Y -129.6058,Z 170,A -101.2922,B 9.96,C 0.3345,E1 9.9301,E2 192.3171} C_DIS
LIN {X -32.9606,Y -128.7859,Z 170,A -102.8394,B 9.96,C 0.3345,E1 9.9259,E2 193.87} C_DIS
LIN {X -38.905,Y -127.1162,Z 170,A -105.5275,B 9.9601,C 0.3333,E1 9.9187,E2 196.5619} C_DIS
LIN {X -42.4876,Y -125.965,Z 170,A -107.0744,B 9.9602,C 0.3305,E1 9.9146,E2 198.1} C_DIS
LIN {X -45.5602,Y -124.8864,Z 170,A -108.6975,B 9.9601,C 0.3336,E1 9.9102,E2 199.7499} C_DIS
LIN {X -49.6572,Y -123.3137,Z 170,A -110.418,B 9.9603,C 0.3284,E1 9.9058,E2 201.4497} C_DIS
LIN {X -52.899,Y -121.9582,Z 170,A -111.9104,B 9.9603,C 0.3264,E1 9.902,E2 202.9395} C_DIS
LIN {X -55.8164,Y -120.6508,Z 170,A -114.2921,B 9.9597,C 0.3445,E1 9.8957,E2 205.4421} C_DIS
LIN {X -61.8761,Y -117.6581,Z 170,A -116.1085,B 9.9606,C 0.3197,E1 9.8915,E2 207.1265} C_DIS
LIN {X -64.152,Y -116.4355,Z 170,A -117.4983,B 9.9604,C 0.3236,E1 9.888,E2 208.5499} C_DIS
LIN {X -67.7482,Y -114.3806,Z 170,A -119.2573,B 9.9605,C 0.3207,E1 9.8837,E2 210.3056} C_DIS
LIN {X -71.4451,Y -112.1083,Z 170,A -121.1699,B 9.9605,C 0.3188,E1 9.8792,E2 212.2231} C_DIS
LIN {X -76.0013,Y -109.0707,Z 170,A -123.4393,B 9.9608,C 0.3134,E1 9.874,E2 214.4811} C_DIS
LIN {X -79.0315,Y -106.8962,Z 170,A -125.1511,B 9.9608,C 0.3128,E1 9.8701,E2 216.2052} C_DIS
LIN {X -82.5373,Y -104.2128,Z 170,A -127.1116,B 9.9608,C 0.3107,E1 9.8658,E2 218.1722} C_DIS
LIN {X -85.1,Y -102.1311,Z 170,A -128.5267,B 9.9609,C 0.308,E1 9.8627,E2 219.586} C_DIS
LIN {X -88.4566,Y -99.2378,Z 170,A -130.4504,B 9.961,C 0.3047,E1 9.8587,E2 221.5108} C_DIS
LIN {X -91.6599,Y -96.2868,Z 170,A -132.3491,B 9.9611,C 0.3016,E1 9.8548,E2 223.4115} C_DIS
LIN {X -94.3057,Y -93.6965,Z 170,A -133.9293,B 9.9612,C 0.2981,E1 9.8517,E2 224.9892} C_DIS
LIN {X -97.5993,Y -90.2615,Z 170,A -136.0046,B 9.9613,C 0.2944,E1 9.8477,E2 227.0666} C_DIS
LIN {X -100.4844,Y -87.0381,Z 170,A -137.7812,B 9.9615,C 0.2888,E1 9.8444,E2 228.8319} C_DIS
LIN {X -102.9275,Y -84.1341,Z 170,A -139.6,B 9.9615,C 0.2886,E1 9.8412,E2 230.6719} C_DIS
LIN {X -105.863,Y -80.4101,Z 170,A -141.6198,B 9.9616,C 0.2836,E1 9.8377,E2 232.6878} C_DIS
LIN {X -108.0827,Y -77.3999,Z 170,A -143.2008,B 9.9618,C 0.2793,E1 9.8351,E2 234.2643} C_DIS
LIN {X -110.3111,Y -74.1904,Z 170,A -144.9557,B 9.9618,C 0.2767,E1 9.8323,E2 236.0268} C_DIS
LIN {X -112.3601,Y -71.048,Z 170,A -146.5242,B 9.962,C 0.2719,E1 9.83,E2 237.5886} C_DIS
LIN {X -114.4464,Y -67.637,Z 170,A -148.3083,B 9.962,C 0.2688,E1 9.8274,E2 239.3789} C_DIS
LIN {X -116.7985,Y -63.4882,Z 170,A -150.4106,B 9.9622,C 0.2645,E1 9.8246,E2 241.4855} C_DIS
LIN {X -118.5353,Y -60.1788,Z 170,A -151.9539,B 9.9622,C 0.2592,E1 9.8226,E2 243.0196} C_DIS
LIN {X -119.9952,Y -57.2122,Z 170,A -153.5419,B 9.9623,C 0.2584,E1 9.8206,E2 244.6261} C_DIS
LIN {X -121.5642,Y -53.8005,Z 170,A -155.0141,B 9.9625,C 0.2516,E1 9.819,E2 246.0798} C_DIS
LIN {X -122.6384,Y -51.3022,Z 170,A -156.2541,B 9.9625,C 0.2497,E1 9.8176,E2 247.327} C_DIS
LIN {X -123.9616,Y -48.017,Z 170,A -157.7633,B 9.9626,C 0.2453,E1 9.8161,E2 248.833} C_DIS
LIN {X -125.193,Y -44.7099,Z 170,A -159.295,B 9.9627,C 0.2413,E1 9.8146,E2 250.3649} C_DIS
LIN {X -126.2593,Y -41.6037,Z 170,A -160.8082,B 9.9627,C 0.2392,E1 9.8132,E2 251.8887} C_DIS
LIN {X -127.5673,Y -37.3992,Z 170,A -163.0504,B 9.9627,C 0.24,E1 9.8114,E2 254.1702} C_DIS
LIN {X -128.5458,Y -33.8858,Z 170,A -164.4883,B 9.9629,C 0.2333,E1 9.8104,E2 255.5909} C_DIS
LIN {X -129.4289,Y -30.346,Z 170,A -165.9818,B 9.9631,C 0.2275,E1 9.8094,E2 257.0739} C_DIS
LIN {X -130.2775,Y -26.4564,Z 170,A -168.5796,B 9.9628,C 0.2379,E1 9.808,E2 259.7741} C_DIS
LIN {X -131.4444,Y -19.8691,Z 170,A -170.3495,B 9.9634,C 0.2103,E1 9.8072,E2 261.4101} C_DIS
LIN {X -131.8229,Y -17.1734,Z 170,A -171.697,B 9.9634,C 0.21,E1 9.8067,E2 262.7772} C_DIS
LIN {X -132.2234,Y -13.7618,Z 170,A -173.3323,B 9.9634,C 0.2084,E1 9.8062,E2 264.4296} C_DIS
LIN {X -132.6159,Y -9.2426,Z 170,A -175.3461,B 9.9636,C 0.2038,E1 9.8057,E2 266.4485} C_DIS
LIN {X -132.8512,Y -4.7888,Z 170,A -177.1301,B 9.9637,C 0.1958,E1 9.8055,E2 268.2142} C_DIS
LIN {X -132.9343,Y -0.986,Z 170,A -178.8818,B 9.9637,C 0.193,E1 9.8055,E2 269.9777} C_DIS
LIN {X -132.8941,Y 3.3881,Z 170,A 179.1595,B 9.9639,C 0.1887,E1 9.8055,E2 271.9432} C_DIS
LIN {X -132.7246,Y 7.5374,Z 170,A 177.3267,B 9.9639,C 0.1843,E1 9.8058,E2 273.7794} C_DIS
LIN {X -132.4557,Y 11.3003,Z 170,A 175.778,B 9.9641,C 0.1782,E1 9.8061,E2 275.3172} C_DIS
LIN {X -132.0701,Y 15.1663,Z 170,A 173.9858,B 9.9641,C 0.1754,E1 9.8066,E2 277.1216} C_DIS
LIN {X -131.5474,Y 19.173,Z 170,A 172.3493,B 9.9642,C 0.1685,E1 9.8073,E2 278.744} C_DIS
LIN {X -130.3202,Y 26.2463,Z 170,A 169.4052,B 9.9644,C 0.157,E1 9.8087,E2 281.6672} C_DIS
LIN {X -129.2539,Y 31.0739,Z 170,A 166.9851,B 9.9644,C 0.1559,E1 9.8102,E2 284.1192} C_DIS
LIN {X -128.3352,Y 34.6755,Z 170,A 165.3965,B 9.9644,C 0.1511,E1 9.8113,E2 285.7046} C_DIS
LIN {X -127.519,Y 37.5644,Z 170,A 164.0739,B 9.9645,C 0.148,E1 9.8123,E2 287.0291} C_DIS
LIN {X -126.5611,Y 40.6749,Z 170,A 162.6541,B 9.9645,C 0.1443,E1 9.8135,E2 288.4494} C_DIS
LIN {X -125.3995,Y 44.1299,Z 170,A 160.9355,B 9.9646,C 0.1426,E1 9.8151,E2 290.1838} C_DIS
LIN {X -123.6213,Y 48.8926,Z 170,A 158.8518,B 9.9647,C 0.1347,E1 9.8172,E2 292.2525} C_DIS
LIN {X -122.4573,Y 51.7359,Z 170,A 157.5067,B 9.9647,C 0.1314,E1 9.8186,E2 293.5986} C_DIS
LIN {X -121.065,Y 54.9167,Z 170,A 155.9952,B 9.9648,C 0.1277,E1 9.8203,E2 295.1103} C_DIS
LIN {X -119.912,Y 57.3864,Z 170,A 154.7082,B 9.9648,C 0.1265,E1 9.8219,E2 296.4092} C_DIS
LIN {X -118.3037,Y 60.6336,Z 170,A 153.172,B 9.9648,C 0.1219,E1 9.8238,E2 297.9407} C_DIS
LIN {X -115.8988,Y 65.116,Z 170,A 150.775,B 9.9649,C 0.1199,E1 9.827,E2 300.3593} C_DIS
LIN {X -113.9028,Y 68.548,Z 170,A 149.263,B 9.965,C 0.112,E1 9.8292,E2 301.8462} C_DIS
LIN {X -111.9459,Y 71.6988,Z 170,A 147.5397,B 9.965,C 0.1102,E1 9.8317,E2 303.5824} C_DIS
LIN {X -109.5981,Y 75.2387,Z 170,A 145.0645,B 9.965,C 0.1172,E1 9.8358,E2 306.1308} C_DIS
LIN {X -106.5052,Y 79.5569,Z 170,A 143.6072,B 9.9652,C 0.097,E1 9.838,E2 307.4886} C_DIS
LIN {X -104.635,Y 82.0009,Z 170,A 142.0091,B 9.9652,C 0.0987,E1 9.8408,E2 309.1172} C_DIS
LIN {X -101.7049,Y 85.6082,Z 170,A 140.0222,B 9.9652,C 0.0939,E1 9.8443,E2 311.1002} C_DIS
LIN {X -99.027,Y 88.692,Z 170,A 138.2074,B 9.9652,C 0.0909,E1 9.8477,E2 312.9195} C_DIS
LIN {X -95.866,Y 92.1001,Z 170,A 136.1798,B 9.9652,C 0.087,E1 9.8516,E2 314.9478} C_DIS
LIN {X -92.7832,Y 95.2053,Z 170,A 134.225,B 9.9652,C 0.0844,E1 9.8554,E2 316.9088} C_DIS
LIN {X -89.5934,Y 98.2128,Z 170,A 132.3559,B 9.9653,C 0.0802,E1 9.8593,E2 318.7737} C_DIS
LIN {X -86.2441,Y 101.1661,Z 170,A 130.5905,B 9.9653,C 0.0735,E1 9.8629,E2 320.5185} C_DIS
LIN {X -83.5165,Y 103.4292,Z 170,A 128.5426,B 9.9653,C 0.0802,E1 9.8675,E2 322.6257} C_DIS
LIN {X -80.439,Y 105.8405,Z 170,A 126.5287,B 9.9653,C 0.0831,E1 9.8721,E2 324.6761} C_DIS
LIN {X -75.9912,Y 109.0777,Z 170,A 124.8034,B 9.9654,C 0.0672,E1 9.8758,E2 326.3242} C_DIS
LIN {X -71.7435,Y 111.9173,Z 170,A 122.5853,B 9.9654,C 0.0639,E1 9.881,E2 328.5422} C_DIS
LIN {X -68.2042,Y 114.1088,Z 170,A 120.7933,B 9.9654,C 0.0611,E1 9.8853,E2 330.3323} C_DIS
LIN {X -65.0897,Y 115.9135,Z 170,A 119.2363,B 9.9654,C 0.0589,E1 9.8891,E2 331.8885} C_DIS
LIN {X -61.5091,Y 117.8508,Z 170,A 117.5095,B 9.9654,C 0.0559,E1 9.8933,E2 333.6105} C_DIS
LIN {X -57.9152,Y 119.6594,Z 170,A 115.8386,B 9.9654,C 0.0524,E1 9.8975,E2 335.2726} C_DIS
LIN {X -55.0624,Y 120.9994,Z 170,A 114.415,B 9.9654,C 0.0519,E1 9.9011,E2 336.7028} C_DIS
LIN {X -52.1008,Y 122.3033,Z 170,A 112.5397,B 9.9654,C 0.0594,E1 9.906,E2 338.6329} C_DIS
LIN {X -48.4292,Y 123.8014,Z 170,A 111.2368,B 9.9655,C 0.0498,E1 9.9093,E2 339.8871} C_DIS
LIN {X -44.8818,Y 125.131,Z 170,A 109.6139,B 9.9655,C 0.0479,E1 9.9135,E2 341.5077} C_DIS
LIN {X -41.8144,Y 126.1892,Z 170,A 108.1933,B 9.9655,C 0.0469,E1 9.9173,E2 342.9298} C_DIS
LIN {X -37.7191,Y 127.4737,Z 170,A 105.955,B 9.9655,C 0.0528,E1 9.9234,E2 345.212} C_DIS
LIN {X -34.0133,Y 128.5118,Z 170,A 104.6762,B 9.9655,C 0.0441,E1 9.9267,E2 346.4453} C_DIS
LIN {X -29.8483,Y 129.5426,Z 170,A 102.8283,B 9.9655,C 0.0428,E1 9.9317,E2 348.2919} C_DIS
LIN {X -26.5994,Y 130.2484,Z 170,A 101.4284,B 9.9655,C 0.0412,E1 9.9356,E2 349.687} C_DIS
LIN {X -22.7174,Y 130.9832,Z 170,A 99.5908,B 9.9655,C 0.0429,E1 9.9406,E2 351.5394} C_DIS
LIN {X -18.6041,Y 131.6287,Z 170,A 97.8813,B 9.9655,C 0.0404,E1 9.9453,E2 353.2377} C_DIS
LIN {X -14.4067,Y 132.154,Z 170,A 96.0743,B 9.9655,C 0.0394,E1 9.9503,E2 355.0418} C_DIS
LIN {X -11.134,Y 132.4698,Z 170,A 94.6698,B 9.9655,C 0.0387,E1 9.9542,E2 356.4441} C_DIS
LIN {X -7.4235,Y 132.7316,Z 170,A 92.9993,B 9.9655,C 0.0397,E1 9.9589,E2 358.1218} C_DIS
LIN {X -3.7253,Y 132.8847,Z 170,A 91.4481,B 9.9655,C 0.0386,E1 9.9632,E2 359.6669} C_DIS
LIN {X 0.3107,Y 132.9373,Z 170,A 89.6066,B 9.9655,C 0.0406,E1 9.9684,E2 361.5196} C_DIS
LIN {X 4.0307,Y 132.8762,Z 170,A 88.0001,B 9.9655,C 0.0407,E1 9.9729,E2 363.1257} C_DIS
LIN {X 8.3698,Y 132.6733,Z 170,A 86.1699,B 9.9655,C 0.0401,E1 9.978,E2 364.9502} C_DIS
LIN {X 12.806,Y 132.3186,Z 170,A 84.3467,B 9.9655,C 0.0385,E1 9.983,E2 366.7616} C_DIS
LIN {X 16.2002,Y 131.9468,Z 170,A 82.856,B 9.9655,C 0.0394,E1 9.9872,E2 368.254} C_DIS
LIN {X 20.2559,Y 131.3845,Z 170,A 81.0771,B 9.9655,C 0.0404,E1 9.9921,E2 370.034} C_DIS
LIN {X 24.1667,Y 130.7238,Z 170,A 79.4198,B 9.9655,C 0.0401,E1 9.9966,E2 371.6847} C_DIS
LIN {X 26.9543,Y 130.1761,Z 170,A 78.2135,B 9.9655,C 0.0404,E1 9.9999,E2 372.8886} C_DIS
LIN {X 29.9104,Y 129.5284,Z 170,A 76.8519,B 9.9655,C 0.0423,E1 10.0036,E2 374.2566} C_DIS
LIN {X 35.8092,Y 128.0228,Z 170,A 74.2315,B 9.9655,C 0.0441,E1 10.0107,E2 376.8761} C_DIS
LIN {X 39.2488,Y 127.011,Z 170,A 72.7198,B 9.9655,C 0.0447,E1 10.0147,E2 378.3835} C_DIS
LIN {X 42.4289,Y 125.9845,Z 170,A 71.1556,B 9.9655,C 0.0486,E1 10.0189,E2 379.9621} C_DIS
LIN {X 45.4598,Y 124.9226,Z 170,A 69.8623,B 9.9655,C 0.0479,E1 10.0223,E2 381.2446} C_DIS
LIN {X 49.9412,Y 123.1992,Z 170,A 67.8532,B 9.9655,C 0.0488,E1 10.0275,E2 383.2465} C_DIS
LIN {X 53.1961,Y 121.8298,Z 170,A 66.342,B 9.9655,C 0.0502,E1 10.0314,E2 384.7564} C_DIS
LIN {X 56.0233,Y 120.5551,Z 170,A 65.0266,B 9.9655,C 0.0513,E1 10.0347,E2 386.0692} C_DIS
LIN {X 59.0724,Y 119.0908,Z 170,A 63.5103,B 9.9655,C 0.0544,E1 10.0385,E2 387.5924} C_DIS
LIN {X 63.2354,Y 116.936,Z 170,A 61.5617,B 9.9655,C 0.0556,E1 10.0433,E2 389.5328} C_DIS
LIN {X 66.0958,Y 115.3431,Z 170,A 60.0689,B 9.9655,C 0.0593,E1 10.047,E2 391.0353} C_DIS
LIN {X 69.5292,Y 113.3062,Z 170,A 58.3633,B 9.9655,C 0.0615,E1 10.0511,E2 392.7393} C_DIS
LIN {X 75.9188,Y 109.1281,Z 170,A 55.1201,B 9.9655,C 0.0657,E1 10.0586,E2 395.9775} C_DIS
LIN {X 79.135,Y 106.8193,Z 170,A 53.3549,B 9.9654,C 0.0699,E1 10.0626,E2 397.7501} C_DIS
LIN {X 81.7561,Y 104.827,Z 170,A 51.9754,B 9.9654,C 0.0715,E1 10.0656,E2 399.1252} C_DIS
LIN {X 85.1607,Y 102.0804,Z 170,A 50.1048,B 9.9654,C 0.0746,E1 10.0697,E2 400.9946} C_DIS
LIN {X 89.7433,Y 98.0757,Z 170,A 47.6282,B 9.9654,C 0.0763,E1 10.0748,E2 403.4546} C_DIS
LIN {X 92.0262,Y 95.9367,Z 170,A 46.1735,B 9.9654,C 0.0813,E1 10.0778,E2 404.9224} C_DIS
LIN {X 96.8227,Y 91.0934,Z 170,A 43.3434,B 9.9653,C 0.0849,E1 10.0833,E2 407.7408} C_DIS
LIN {X 99.6399,Y 88.0028,Z 170,A 41.5135,B 9.9653,C 0.0894,E1 10.0867,E2 409.5747} C_DIS
LIN {X 104.4567,Y 82.2278,Z 170,A 38.2884,B 9.9652,C 0.0962,E1 10.0924,E2 412.7995} C_DIS
LIN {X 107.2458,Y 78.5556,Z 170,A 36.1567,B 9.9651,C 0.1042,E1 10.096,E2 414.9492} C_DIS
LIN {X 110.2231,Y 74.3205,Z 170,A 34.114,B 9.9651,C 0.1051,E1 10.0992,E2 416.9707} C_DIS
LIN {X 112.6098,Y 70.6525,Z 170,A 32.2531,B 9.9651,C 0.1091,E1 10.102,E2 418.8298} C_DIS
LIN {X 114.8057,Y 67.0254,Z 170,A 30.0082,B 9.9649,C 0.1233,E1 10.1053,E2 421.1253} C_DIS
LIN {X 117.0181,Y 63.0822,Z 170,A 28.5793,B 9.9649,C 0.1162,E1 10.1071,E2 422.4937} C_DIS
LIN {X 118.6219,Y 60.0087,Z 170,A 27.117,B 9.9649,C 0.1193,E1 10.1089,E2 423.9532} C_DIS
LIN {X 120.2838,Y 56.6082,Z 170,A 25.5525,B 9.9649,C 0.122,E1 10.1108,E2 425.5108} C_DIS
LIN {X 121.4384,Y 54.0819,Z 170,A 24.3923,B 9.9649,C 0.1242,E1 10.1121,E2 426.6674} C_DIS
LIN {X 122.7148,Y 51.1193,Z 170,A 22.9921,B 9.9649,C 0.1282,E1 10.1137,E2 428.0698} C_DIS
LIN {X 124.6225,Y 46.2761,Z 170,A 20.7915,B 9.9647,C 0.1332,E1 10.1159,E2 430.2669} C_DIS
LIN {X 125.6467,Y 43.4169,Z 170,A 19.4843,B 9.9647,C 0.1368,E1 10.1171,E2 431.5749} C_DIS
LIN {X 126.9083,Y 39.5842,Z 170,A 17.2955,B 9.9645,C 0.1522,E1 10.119,E2 433.8188} C_DIS
LIN {X 128.0654,Y 35.6568,Z 170,A 16.0089,B 9.9645,C 0.1458,E1 10.1199,E2 435.0497} C_DIS
LIN {X 129.1074,Y 31.6817,Z 170,A 14.2136,B 9.9645,C 0.1514,E1 10.1212,E2 436.8495} C_DIS
LIN {X 129.9378,Y 28.077,Z 170,A 12.6972,B 9.9645,C 0.154,E1 10.1221,E2 438.3578} C_DIS
LIN {X 130.6864,Y 24.3637,Z 170,A 10.9844,B 9.9643,C 0.1606,E1 10.123,E2 440.0818} C_DIS
LIN {X 131.3664,Y 20.3724,Z 170,A 9.3909,B 9.9643,C 0.162,E1 10.1237,E2 441.6586} C_DIS
LIN {X 131.8331,Y 17.0956,Z 170,A 7.989,B 9.9643,C 0.1655,E1 10.1242,E2 443.0588} C_DIS
LIN {X 132.2418,Y 13.591,Z 170,A 6.3504,B 9.9641,C 0.1727,E1 10.1247,E2 444.713} C_DIS
LIN {X 132.5924,Y 9.5645,Z 170,A 4.7317,B 9.9641,C 0.1749,E1 10.1251,E2 446.3185} C_DIS
LIN {X 132.8303,Y 5.326,Z 170,A 2.9583,B 9.9641,C 0.1788,E1 10.1253,E2 448.0868} C_DIS
LIN {X 132.9248,Y 1.8357,Z 170,A 1.4637,B 9.964,C 0.183,E1 10.1254,E2 449.5817} C_DIS
LIN {X 132.9123,Y -2.5853,Z 170,A -0.3806,B 9.9639,C 0.1871,E1 10.1254,E2 451.4205} C_DIS
LIN {X 132.8059,Y -5.9454,Z 170,A -1.9702,B 9.9637,C 0.1947,E1 10.1252,E2 453.0286} C_DIS
LIN {X 132.5706,Y -9.8627,Z 170,A -3.5383,B 9.9637,C 0.1967,E1 10.1249,E2 454.5834} C_DIS
LIN {X 132.1915,Y -14.0579,Z 170,A -5.2819,B 9.9637,C 0.2003,E1 10.1244,E2 456.3201} C_DIS
LIN {X 131.8154,Y -17.2303,Z 170,A -6.6305,B 9.9636,C 0.2036,E1 10.124,E2 457.6668} C_DIS
LIN {X 131.3451,Y -20.51,Z 170,A -8.0409,B 9.9635,C 0.2073,E1 10.1234,E2 459.0765} C_DIS
LIN {X 130.6429,Y -24.5916,Z 170,A -9.8986,B 9.9634,C 0.2142,E1 10.1225,E2 460.9449} C_DIS
LIN {X 129.7893,Y -28.765,Z 170,A -12.1327,B 9.963,C 0.229,E1 10.1211,E2 463.229} C_DIS
LIN {X 128.7771,Y -32.9951,Z 170,A -13.7598,B 9.963,C 0.2284,E1 10.12,E2 464.8282} C_DIS
LIN {X 127.9165,Y -36.1891,Z 170,A -14.8355,B 9.9631,C 0.2241,E1 10.1192,E2 465.8631} C_DIS
LIN {X 127.0189,Y -39.2229,Z 170,A -16.2078,B 9.9631,C 0.2282,E1 10.1181,E2 467.2379} C_DIS
LIN {X 125.4033,Y -44.1192,Z 170,A -18.3753,B 9.9629,C 0.2331,E1 10.1162,E2 469.4013} C_DIS
LIN {X 124.3611,Y -46.9739,Z 170,A -19.6832,B 9.9629,C 0.2367,E1 10.1149,E2 470.7103} C_DIS
LIN {X 122.9226,Y -50.6216,Z 170,A -21.4531,B 9.9627,C 0.2433,E1 10.1131,E2 472.4918} C_DIS
LIN {X 120.1582,Y -56.871,Z 170,A -24.122,B 9.9627,C 0.2446,E1 10.1101,E2 475.1304} C_DIS
LIN {X 118.8056,Y -59.6478,Z 170,A -25.6783,B 9.9624,C 0.2535,E1 10.1081,E2 476.7156} C_DIS
LIN {X 116.9028,Y -63.2969,Z 170,A -27.3831,B 9.9624,C 0.2566,E1 10.1059,E2 478.4139} C_DIS
LIN {X 114.0961,Y -68.2255,Z 170,A -29.6729,B 9.9623,C 0.2592,E1 10.1027,E2 480.6876} C_DIS
LIN {X 112.2158,Y -71.2766,Z 170,A -31.3849,B 9.9621,C 0.2671,E1 10.1001,E2 482.4215} C_DIS
LIN {X 109.5334,Y -75.333,Z 170,A -33.179,B 9.9621,C 0.2652,E1 10.0974,E2 484.1812} C_DIS
LIN {X 107.7193,Y -77.9049,Z 170,A -34.7235,B 9.9619,C 0.2729,E1 10.0949,E2 485.75} C_DIS
LIN {X 105.3507,Y -81.0802,Z 170,A -36.4263,B 9.9619,C 0.2769,E1 10.092,E2 487.4542} C_DIS
LIN {X 102.883,Y -84.1885,Z 170,A -38.9095,B 9.9612,C 0.2989,E1 10.0874,E2 490.0325} C_DIS
LIN {X 98.8124,Y -88.9315,Z 170,A -40.8897,B 9.9615,C 0.2884,E1 10.0839,E2 491.9295} C_DIS
LIN {X 95.6748,Y -92.2984,Z 170,A -42.7877,B 9.9615,C 0.2908,E1 10.0803,E2 493.8191} C_DIS
LIN {X 89.8098,Y -98.0146,Z 170,A -45.9116,B 9.9615,C 0.2888,E1 10.0741,E2 496.8971} C_DIS
LIN {X 87.1465,Y -100.3903,Z 170,A -47.7676,B 9.9612,C 0.2993,E1 10.0701,E2 498.7935} C_DIS
LIN {X 83.787,Y -103.2111,Z 170,A -49.8116,B 9.961,C 0.3065,E1 10.0657,E2 500.8581} C_DIS
LIN {X 80.9218,Y -105.4718,Z 170,A -51.2242,B 9.961,C 0.3058,E1 10.0626,E2 502.2527} C_DIS
LIN {X 77.3423,Y -108.1239,Z 170,A -53.2098,B 9.9608,C 0.3108,E1 10.0581,E2 504.2481} C_DIS
LIN {X 74.2747,Y -110.2541,Z 170,A -54.7396,B 9.9608,C 0.3118,E1 10.0546,E2 505.7698} C_DIS
LIN {X 70.488,Y -112.7126,Z 170,A -56.9709,B 9.9605,C 0.3215,E1 10.0492,E2 508.0376} C_DIS
LIN {X 67.1193,Y -114.7505,Z 170,A -58.445,B 9.9605,C 0.3191,E1 10.0457,E2 509.4861} C_DIS
LIN {X 63.3114,Y -116.895,Z 170,A -60.2466,B 9.9605,C 0.3201,E1 10.0413,E2 511.2795} C_DIS
LIN {X 58.4506,Y -119.3975,Z 170,A -62.4154,B 9.9605,C 0.3193,E1 10.036,E2 513.4274} C_DIS
LIN {X 55.5296,Y -120.7834,Z 170,A -63.8197,B 9.9605,C 0.3214,E1 10.0324,E2 514.8342} C_DIS
LIN {X 52.1246,Y -122.293,Z 170,A -65.4081,B 9.9605,C 0.3231,E1 10.0284,E2 516.4219} C_DIS
LIN {X 46.8858,Y -124.3941,Z 170,A -67.9227,B 9.9603,C 0.3278,E1 10.0218,E2 518.9483} C_DIS
LIN {X 41.8362,Y -126.1819,Z 170,A -70.1268,B 9.9603,C 0.3279,E1 10.016,E2 521.1415} C_DIS
LIN {X 38.9111,Y -127.1143,Z 170,A -71.599,B 9.9601,C 0.3325,E1 10.012,E2 522.6329} C_DIS
LIN {X 34.4925,Y -128.384,Z 170,A -73.431,B 9.9601,C 0.331,E1 10.0072,E2 524.4481} C_DIS
LIN {X 30.9968,Y -129.2724,Z 170,A -74.9717,B 9.9601,C 0.332,E1 10.003,E2 525.9882} C_DIS
LIN {X 27.6083,Y -130.039,Z 170,A -76.5664,B 9.9601,C 0.3352,E1 9.9986,E2 527.5958} C_DIS
LIN {X 23.4909,Y -130.8448,Z 170,A -78.2833,B 9.9601,C 0.3344,E1 9.9939,E2 529.3027} C_DIS
LIN {X 19.5165,Y -131.4983,Z 170,A -80.1223,B 9.96,C 0.3377,E1 9.9888,E2 531.1554} C_DIS
LIN {X 15.3928,Y -132.0431,Z 170,A -81.8853,B 9.96,C 0.3379,E1 9.9839,E2 532.9158} C_DIS
LIN {X 11.1587,Y -132.4677,Z 170,A -83.6052,B 9.96,C 0.3362,E1 9.9792,E2 534.6227} C_DIS
LIN {X 7.4012,Y -132.7324,Z 170,A -85.3359,B 9.96,C 0.339,E1 9.9743,E2 536.3675} C_DIS
LIN {X 3.2388,Y -132.8982,Z 170,A -86.9948,B 9.96,C 0.3365,E1 9.9697,E2 538.0106} C_DIS
LIN {X 0.9614,Y -132.9326,Z 170,A -87.8087,B 9.9601,C 0.3331,E1 9.9675,E2 538.8044} C_DIS
Enddeposition()
LIN {X 0.9614,Y -132.9326,Z 170,A -87.8087,B 9.9601,C 0.3331,E1 9.9675,E2 538.8044} C_DIS
Startdeposition()
$VEL.CP = VEL_PRINT
LIN {X 2.045,Y -133.8332,Z 170,A -86.7893,B 9.9602,C 0.327,E1 9.9704,E2 537.7504} C_DIS
LIN {X 5.7086,Y -133.7278,Z 170,A -84.9609,B 9.9604,C 0.321,E1 9.9755,E2 535.8888} C_DIS
LIN {X 9.1782,Y -133.5348,Z 170,A -83.7449,B 9.9602,C 0.3264,E1 9.9788,E2 534.7059} C_DIS
LIN {X 12.7336,Y -133.2415,Z 170,A -82.2167,B 9.9602,C 0.3258,E1 9.9831,E2 533.1767} C_DIS
LIN {X 17.0919,Y -132.7531,Z 170,A -80.4153,B 9.9602,C 0.3266,E1 9.9881,E2 531.3837} C_DIS
LIN {X 20.4274,Y -132.2806,Z 170,A -78.978,B 9.9602,C 0.3259,E1 9.992,E2 529.9461} C_DIS
LIN {X 23.8222,Y -131.7117,Z 170,A -77.4908,B 9.9602,C 0.3247,E1 9.9961,E2 528.4562} C_DIS
LIN {X 27.872,Y -130.9149,Z 170,A -75.7307,B 9.9603,C 0.3236,E1 10.001,E2 526.6959} C_DIS
LIN {X 31.3602,Y -130.1227,Z 170,A -74.2147,B 9.9603,C 0.3227,E1 10.0051,E2 525.1806} C_DIS
LIN {X 34.8505,Y -129.2322,Z 170,A -72.7402,B 9.9603,C 0.3229,E1 10.009,E2 523.7135} C_DIS
LIN {X 38.2663,Y -128.2635,Z 170,A -71.0705,B 9.9605,C 0.3181,E1 10.0136,E2 522.0241} C_DIS
LIN {X 42.8528,Y -126.8044,Z 170,A -68.8662,B 9.9607,C 0.3127,E1 10.0195,E2 519.8001} C_DIS
LIN {X 47.8745,Y -124.9944,Z 170,A -66.9483,B 9.9605,C 0.3185,E1 10.0244,E2 517.9263} C_DIS
LIN {X 51.3844,Y -123.5922,Z 170,A -65.2282,B 9.9606,C 0.3142,E1 10.0289,E2 516.1921} C_DIS
LIN {X 54.4451,Y -122.2747,Z 170,A -63.8257,B 9.9606,C 0.3129,E1 10.0324,E2 514.7914} C_DIS
LIN {X 57.1877,Y -121.0174,Z 170,A -62.3656,B 9.9608,C 0.3073,E1 10.0362,E2 513.3092} C_DIS
LIN {X 61.6043,Y -118.8306,Z 170,A -60.4442,B 9.9608,C 0.3086,E1 10.0409,E2 511.4095} C_DIS
LIN {X 66.6788,Y -116.0587,Z 170,A -57.7678,B 9.9611,C 0.3002,E1 10.0475,E2 508.7057} C_DIS
LIN {X 70.9706,Y -113.4862,Z 170,A -55.7698,B 9.9611,C 0.3,E1 10.0522,E2 506.7238} C_DIS
LIN {X 74.6788,Y -111.0816,Z 170,A -54.0902,B 9.9611,C 0.3018,E1 10.0561,E2 505.0689} C_DIS
LIN {X 79.3687,Y -107.7798,Z 170,A -51.7474,B 9.9611,C 0.3,E1 10.0614,E2 502.7378} C_DIS
LIN {X 83.7628,Y -104.4019,Z 170,A -49.0889,B 9.9614,C 0.2888,E1 10.0674,E2 500.0415} C_DIS
LIN {X 87.2398,Y -101.514,Z 170,A -47.2013,B 9.9614,C 0.2861,E1 10.0714,E2 498.1578} C_DIS
LIN {X 90.5953,Y -98.531,Z 170,A -45.5753,B 9.9614,C 0.2892,E1 10.0747,E2 496.5667} C_DIS
LIN {X 93.1087,Y -96.1593,Z 170,A -43.7944,B 9.9617,C 0.2789,E1 10.0783,E2 494.7467} C_DIS
LIN {X 96.4018,Y -92.8582,Z 170,A -41.897,B 9.9617,C 0.277,E1 10.082,E2 492.8596} C_DIS
LIN {X 99.2532,Y -89.8037,Z 170,A -40.2064,B 9.9617,C 0.2753,E1 10.0852,E2 491.1793} C_DIS
LIN {X 102.0697,Y -86.589,Z 170,A -38.2185,B 9.962,C 0.2674,E1 10.0889,E2 489.1698} C_DIS
LIN {X 105.0572,Y -82.9394,Z 170,A -36.4591,B 9.962,C 0.2688,E1 10.0919,E2 487.4405} C_DIS
LIN {X 107.6878,Y -79.494,Z 170,A -34.5187,B 9.9621,C 0.2624,E1 10.0952,E2 485.4876} C_DIS
LIN {X 110.9867,Y -74.8189,Z 170,A -32.0698,B 9.9623,C 0.2564,E1 10.0991,E2 483.0361} C_DIS
LIN {X 113.2579,Y -71.3339,Z 170,A -30.2944,B 9.9623,C 0.252,E1 10.1018,E2 481.2595} C_DIS
LIN {X 114.9484,Y -68.5765,Z 170,A -28.0523,B 9.963,C 0.2276,E1 10.1051,E2 478.9085} C_DIS
LIN {X 118.2561,Y -62.6984,Z 170,A -26.2185,B 9.9625,C 0.2457,E1 10.1074,E2 477.2034} C_DIS
LIN {X 122.0576,Y -54.9305,Z 170,A -22.4044,B 9.9628,C 0.2331,E1 10.112,E2 473.3717} C_DIS
LIN {X 123.6694,Y -51.1996,Z 170,A -20.6805,B 9.9629,C 0.2288,E1 10.1139,E2 471.6478} C_DIS
LIN {X 125.2526,Y -47.1933,Z 170,A -19.0215,B 9.9629,C 0.2282,E1 10.1155,E2 470.0097} C_DIS
LIN {X 126.8126,Y -42.8274,Z 170,A -16.8109,B 9.9632,C 0.2171,E1 10.1176,E2 467.769} C_DIS
LIN {X 128.0183,Y -39.0729,Z 170,A -14.8048,B 9.9635,C 0.2046,E1 10.1193,E2 465.7215} C_DIS
LIN {X 129.2859,Y -34.6486,Z 170,A -13.1266,B 9.9635,C 0.2061,E1 10.1205,E2 464.0775} C_DIS
LIN {X 130.0816,Y -31.5307,Z 170,A -11.9922,B 9.9634,C 0.2081,E1 10.1212,E2 462.9718} C_DIS
LIN {X 130.9568,Y -27.6777,Z 170,A -10.2589,B 9.9635,C 0.2023,E1 10.1222,E2 461.2316} C_DIS
LIN {X 131.7147,Y -23.8057,Z 170,A -8.6664,B 9.9635,C 0.1997,E1 10.123,E2 459.6492} C_DIS
LIN {X 132.3387,Y -20.0516,Z 170,A -6.9881,B 9.9637,C 0.1938,E1 10.1238,E2 457.9632} C_DIS
LIN {X 132.9045,Y -15.8691,Z 170,A -5.3159,B 9.9637,C 0.1918,E1 10.1244,E2 456.3056} C_DIS
LIN {X 133.3112,Y -12.0047,Z 170,A -3.5948,B 9.9638,C 0.1856,E1 10.1248,E2 454.5758} C_DIS
LIN {X 133.6357,Y -7.5753,Z 170,A -1.7032,B 9.9639,C 0.1803,E1 10.1252,E2 452.6834} C_DIS
LIN {X 133.7977,Y -3.6955,Z 170,A -0.1654,B 9.9639,C 0.1784,E1 10.1253,E2 451.1593} C_DIS
LIN {X 133.8497,Y 0.3583,Z 170,A 1.6135,B 9.9641,C 0.1723,E1 10.1253,E2 449.3734} C_DIS
LIN {X 133.7764,Y 4.4612,Z 170,A 3.3269,B 9.9641,C 0.1682,E1 10.1253,E2 447.6637} C_DIS
LIN {X 133.596,Y 8.2197,Z 170,A 4.8479,B 9.9641,C 0.1657,E1 10.125,E2 446.152} C_DIS
LIN {X 133.3126,Y 11.9882,Z 170,A 6.4742,B 9.9642,C 0.1608,E1 10.1246,E2 444.5232} C_DIS
LIN {X 132.899,Y 15.9149,Z 170,A 8.1518,B 9.9643,C 0.1562,E1 10.1241,E2 442.8456} C_DIS
LIN {X 132.3268,Y 20.1288,Z 170,A 9.9535,B 9.9643,C 0.1514,E1 10.1234,E2 441.0445} C_DIS
LIN {X 131.7133,Y 23.8134,Z 170,A 11.5015,B 9.9644,C 0.1481,E1 10.1226,E2 439.5013} C_DIS
LIN {X 130.9132,Y 27.8797,Z 170,A 13.2198,B 9.9644,C 0.1444,E1 10.1217,E2 437.7884} C_DIS
LIN {X 130.107,Y 31.4256,Z 170,A 14.7465,B 9.9646,C 0.1407,E1 10.1207,E2 436.264} C_DIS
LIN {X 129.1632,Y 35.1092,Z 170,A 16.3091,B 9.9646,C 0.1377,E1 10.1196,E2 434.7081} C_DIS
LIN {X 126.7617,Y 42.9809,Z 170,A 19.7899,B 9.9647,C 0.129,E1 10.1167,E2 431.2299} C_DIS
LIN {X 124.3091,Y 49.6265,Z 170,A 22.8119,B 9.9648,C 0.1211,E1 10.1137,E2 428.2069} C_DIS
LIN {X 123.1956,Y 52.334,Z 170,A 24.2209,B 9.9648,C 0.114,E1 10.1122,E2 426.7781} C_DIS
LIN {X 121.6466,Y 55.8351,Z 170,A 25.6699,B 9.9648,C 0.1142,E1 10.1105,E2 425.3511} C_DIS
LIN {X 120.1454,Y 58.9954,Z 170,A 27.1715,B 9.9649,C 0.1102,E1 10.1087,E2 423.848} C_DIS
LIN {X 118.1768,Y 62.8494,Z 170,A 29.0849,B 9.9649,C 0.104,E1 10.1062,E2 421.926} C_DIS
LIN {X 115.3916,Y 67.828,Z 170,A 31.4428,B 9.965,C 0.0999,E1 10.103,E2 419.5768} C_DIS
LIN {X 113.1421,Y 71.5173,Z 170,A 33.3035,B 9.965,C 0.0951,E1 10.1002,E2 417.7138} C_DIS
LIN {X 110.7329,Y 75.1938,Z 170,A 34.938,B 9.965,C 0.0964,E1 10.0978,E2 416.1082} C_DIS
LIN {X 108.4021,Y 78.5166,Z 170,A 36.8639,B 9.9652,C 0.0879,E1 10.0946,E2 414.1586} C_DIS
LIN {X 105.6088,Y 82.2358,Z 170,A 39.3718,B 9.9652,C 0.0712,E1 10.0902,E2 411.5865} C_DIS
LIN {X 102.5267,Y 86.0472,Z 170,A 40.9301,B 9.9652,C 0.0793,E1 10.0875,E2 410.0933} C_DIS
LIN {X 99.503,Y 89.5271,Z 170,A 42.8807,B 9.9652,C 0.0755,E1 10.0839,E2 408.1447} C_DIS
LIN {X 97.0709,Y 92.159,Z 170,A 44.3415,B 9.9652,C 0.074,E1 10.0812,E2 406.6921} C_DIS
LIN {X 94.2831,Y 95.0082,Z 170,A 46.0472,B 9.9652,C 0.0706,E1 10.0778,E2 404.9858} C_DIS
LIN {X 91.2705,Y 97.9058,Z 170,A 47.7185,B 9.9652,C 0.0698,E1 10.0745,E2 403.3282} C_DIS
LIN {X 88.8404,Y 100.1164,Z 170,A 49.2817,B 9.9653,C 0.0635,E1 10.0712,E2 401.7455} C_DIS
LIN {X 85.3084,Y 103.1424,Z 170,A 51.2242,B 9.9653,C 0.0609,E1 10.067,E2 399.8084} C_DIS
LIN {X 82.1699,Y 105.6599,Z 170,A 52.9029,B 9.9653,C 0.0588,E1 10.0633,E2 398.1346} C_DIS
LIN {X 78.841,Y 108.1669,Z 170,A 54.8859,B 9.9654,C 0.0513,E1 10.0588,E2 396.1271} C_DIS
LIN {X 72.8785,Y 112.2702,Z 170,A 57.7335,B 9.9654,C 0.052,E1 10.0523,E2 393.3094} C_DIS
LIN {X 69.4756,Y 114.4075,Z 170,A 59.5298,B 9.9654,C 0.0477,E1 10.048,E2 391.5036} C_DIS
LIN {X 65.6571,Y 116.6406,Z 170,A 61.2923,B 9.9654,C 0.048,E1 10.0438,E2 389.7569} C_DIS
LIN {X 62.5553,Y 118.3313,Z 170,A 62.6675,B 9.9654,C 0.049,E1 10.0404,E2 388.398} C_DIS
LIN {X 60.0091,Y 119.6448,Z 170,A 64.1027,B 9.9654,C 0.0428,E1 10.0368,E2 386.9377} C_DIS
LIN {X 56.4256,Y 121.3736,Z 170,A 65.704,B 9.9654,C 0.043,E1 10.0328,E2 385.3485} C_DIS
LIN {X 53.3997,Y 122.7351,Z 170,A 67.1028,B 9.9654,C 0.0418,E1 10.0292,E2 383.9524} C_DIS
LIN {X 50.4869,Y 123.9623,Z 170,A 68.5894,B 9.9654,C 0.0374,E1 10.0253,E2 382.4497} C_DIS
LIN {X 45.8507,Y 125.7509,Z 170,A 71.0296,B 9.9654,C 0.0285,E1 10.0189,E2 379.9719} C_DIS
LIN {X 41.9017,Y 127.1211,Z 170,A 72.2669,B 9.9654,C 0.039,E1 10.0158,E2 378.8014} C_DIS
LIN {X 34.9899,Y 129.195,Z 170,A 75.4886,B 9.9654,C 0.0337,E1 10.0071,E2 375.5645} C_DIS
LIN {X 31.1004,Y 130.1854,Z 170,A 77.1173,B 9.9654,C 0.0345,E1 10.0027,E2 373.9469} C_DIS
LIN {X 27.1872,Y 131.0592,Z 170,A 78.8862,B 9.9654,C 0.0324,E1 9.9979,E2 372.1722} C_DIS
LIN {X 23.541,Y 131.762,Z 170,A 80.4507,B 9.9654,C 0.0321,E1 9.9936,E2 370.611} C_DIS
LIN {X 19.286,Y 132.4523,Z 170,A 82.2977,B 9.9654,C 0.0313,E1 9.9885,E2 368.7644} C_DIS
LIN {X 15.3363,Y 132.9681,Z 170,A 84.034,B 9.9654,C 0.0301,E1 9.9836,E2 367.025} C_DIS
LIN {X 11.5415,Y 133.3504,Z 170,A 85.6293,B 9.9654,C 0.0305,E1 9.9792,E2 365.4347} C_DIS
LIN {X 7.5604,Y 133.6366,Z 170,A 87.44,B 9.9654,C 0.0281,E1 9.9741,E2 363.6125} C_DIS
LIN {X 3.8771,Y 133.7926,Z 170,A 88.8853,B 9.9654,C 0.0308,E1 9.9702,E2 362.1837} C_DIS
LIN {X 0.2032,Y 133.8497,Z 170,A 90.5989,B 9.9654,C 0.0279,E1 9.9653,E2 360.454} C_DIS
LIN {X -4.1253,Y 133.7857,Z 170,A 92.4253,B 9.9654,C 0.0286,E1 9.9602,E2 358.6317} C_DIS
LIN {X -8.1433,Y 133.6007,Z 170,A 94.0393,B 9.9654,C 0.0312,E1 9.9558,E2 357.0314} C_DIS
LIN {X -12.1077,Y 133.3016,Z 170,A 95.7269,B 9.9654,C 0.0319,E1 9.9511,E2 355.3466} C_DIS
LIN {X -15.7576,Y 132.9178,Z 170,A 97.2348,B 9.9654,C 0.0338,E1 9.9469,E2 353.847} C_DIS
LIN {X -18.8884,Y 132.5091,Z 170,A 98.6537,B 9.9654,C 0.033,E1 9.943,E2 352.4209} C_DIS
LIN {X -22.3236,Y 131.9741,Z 170,A 100.172,B 9.9654,C 0.0331,E1 9.9388,E2 350.8998} C_DIS
LIN {X -25.9931,Y 131.3022,Z 170,A 101.8652,B 9.9654,C 0.0321,E1 9.9341,E2 349.1962} C_DIS
LIN {X -29.7329,Y 130.5042,Z 170,A 103.3395,B 9.9654,C 0.0365,E1 9.9302,E2 347.7424} C_DIS
LIN {X -32.7824,Y 129.7718,Z 170,A 104.698,B 9.9654,C 0.0371,E1 9.9265,E2 346.3829} C_DIS
LIN {X -40.4297,Y 127.5966,Z 170,A 108.2099,B 9.9654,C 0.0379,E1 9.917,E2 342.8607} C_DIS
LIN {X -44.6816,Y 126.1724,Z 170,A 110.8098,B 9.9654,C 0.0264,E1 9.91,E2 340.1804} C_DIS
LIN {X -49.6642,Y 124.2939,Z 170,A 112.5211,B 9.9654,C 0.0401,E1 9.9057,E2 338.5393} C_DIS
LIN {X -53.9397,Y 122.5008,Z 170,A 114.5175,B 9.9654,C 0.0422,E1 9.9006,E2 336.5432} C_DIS
Enddeposition()
END
